(* CODESYS project partidas_v1_9_11.library
   DefaultNamespace: Teknike_Partidas
   DocFormat: reStructuredText
   Description: Bliblioteca com as partidas usadas pela Teknike
   Author: Tiago B. Cunico
   Title: Partidas
   Version: 1.9.11
   Company: Teknike
   Placeholder: Teknike_Partidas

Project tree, tasks and I/O mapping:
  libraries: OSCAT - AixOCAT, * (RWTH Aachen University - E.ON Energy Research Center); Tc2_MC2, * (Beckhoff Automation GmbH); Tc2_MC2_Drive, * (Beckhoff Automation GmbH); Tc2_ModbusRTU, * (Beckhoff Automation GmbH); Tc2_ModbusSrv, * (Beckhoff Automation GmbH); Tc2_Standard, * (Beckhoff Automation GmbH); Tc2_System, * (Beckhoff Automation GmbH); Tc2_Utilities, * (Beckhoff Automation GmbH); Tc3_Database, * (Beckhoff Automation GmbH); Tc3_Module, * (Beckhoff Automation GmbH); TcUnit, * (www.tcunit.org); Geral, * (Teknike)
  Legado/
    function block FB_ATV320CAN_V2_Legado [ST]: ACT_TrabalhaDados, ACT01_LeiturasCAN, ACT03_Cicla, ACT04_WriteCAN
    function block FB_Ethernet_ATV630_V2_Legado [ST]: ACT_00_LeituraETA_CIA402, ACT_01_LeituraVelocidadeAtual, ACT_03_EscritaVelocidade, ACT_04_Leitura_Last_error, ACT_05_LeituraETA_UINT, ACT_06_Leitura_Motor_Therm, ACT_07_Leitura_Motor_run_time, ACT_08_Leitura_Sto_Status, ACT_09_Leitura_APPS, ACT_HearthBeat
    function block FB_PartidaDireta_V2_Legado [ST]
    function block FB_PartidaDiretaReversao_V0_Legado [ST]
  POUs/
    Beckhoff/
      AX5000/
        Sts/
        function block FB_Comunicacao_AX5000 [ST]: ControlaACCDEC, LeParametros, Status
    Comunicação/
      CAN/
        Sts/
          data type ATV320_Can
          data type Config_CAN
          data type Config_CAN_Normal
          data type Config_CAN_Retentiva
          data type MaquinaCanOpen
        TeSys U/
          Sts/
            data type st_IosTeSysU_Can
            data type st_IosTeSysU_Can_IN
            data type st_IosTeSysU_Can_OUT
          function block FB_TeSysU_Can [ST]: AlertasEFalhas, IOs_vista
        function block FB_ComunicacaoCanOpen [ST]: AcaoMaquinaDeEstados, EscritaPDO, Escritas_SDO, Leituras_SDO, Status, TrocaEstadoMaquinaDeEstados
        function block SDO_READ [ST]
        function block SDO_WRITE [ST]
      Ethernet/
        data type ConfigComunicacaoEthernet
        function block ConversaoBilateralConfig [ST]
        function block FB_ComunicacaoEthernet [ST]: AcaoMaquinaDeEstados, Ciclo1s, Escrita, IHM, Leituras, Leituras_Escritas, MaquinaDeEstados, TrocaEstadoMaquinaDeEstados
        data type st_ReadWriteREG
      EthernetIP/
        Delta/
          Sts/
            data type st_LinkDeltaEIP
          function block FB_DeltaMS [ST]: ControleMarcha, ControleVelocidade, Emergencia, Others, Status
      ModbusRTU/
        STs/
          data type State_Modbus
          data type StateWord
        function block FB_ControleSoftRTU_LEGADO [ST]: Status
        function block FB_ModBusRTU_AC380 [ST]: Escrita, EspelhoEntradas, EspelhoSaidas, Estados, ExecutaEstados, Leitura, Leitura_Escrita, Status
        function block FB_ModBusRTU_ALTISTAR22 [ST]: Escrita, EspelhoEntradas, EspelhoSaidas, Estados, ExecutaEstados, Leitura, Leitura_Escrita, Status
        function block FB_ModBusRTU_ATV320 [ST]: Escrita, EspelhoEntradas, EspelhoSaidas, Estados, ExecutaEstados, Leitura, Leitura_Escrita, Status
    Partida/
      Sts/
        data type ST_ConfigInversor
        data type ST_ConfigMotorDB
        data type st_ConfigPartida
        data type st_EntradaPartida
        data type st_Erros
        data type st_KPIPartida
        data type st_LeiturasInversor
        data type st_LeiturasInversorIHM
        data type st_Partida
        data type st_SaidaPartida
      Test/
        function block FB_Partida_Teste [ST]: Bypasses, Emergencia, Falhas, Interlocks, ProxPartida, Reversao, Velocidade
      function block FB_Partida [ST]: AjustaEntradaST, AjustaSaida, AlarmesIHM, Contagem, ControleBloqueio, ControleDaPartida, ControleReset, ControleVelocidade, EmComissionamento, Falhas, FB_init, FirstScan, Horimetro, KPI, ProxMotor, SegurancaReversao, Status
    Siemens/
      Geral/
        data type bits
        data type Bits_8
        data type Duint
        data type Inversor_2Words_SinaSpeed
        data type InversorSinaSpeed
        data type sxRecvBuf
        data type sxSendBuf
        data type u16b
        data type Word_Bits
      SinaSpeed/
        data type EntradaSinaSpeed
        data type SaidaSinaSpeed
        function block Sina_SpeedV2 [ST]
        data type st_SinaSpeed
      function block Sina_posV2 [ST]
    global variables GVL_BlibliotecaPartidas
    program PRG_TEST [ST]: Teste, TesteAX5000, TesteCan, TesteCanTeSysU, TesteDelta, TestePartida, TestePartidaSimples, TesteProfinet
    program ValidaLicensa [ST]: Licensas
  Project Information/
    function F_GetCompany [ST]
    function F_GetTitle [ST]
    function F_GetVersion [ST]
  Version/
    global variables Global_Version
  VISUs/
*)

// POUs/Comunicação/CAN/Sts/ATV320_Can
TYPE ATV320_Can :
	STRUCT
		NodeState AT %I* : USINT;

		StatusWord		AT %I*	: UINT;
		ControlEffort	AT %I*	: INT;
		NM1				AT %I*	: UINT;
		NM2				AT %I*	: UINT;
		NM3				AT %I*	: UINT;
		NM4				AT %I*	: UINT;

		Controlword		AT %Q*	: UINT;
		TargetVelocity	AT %Q*	: INT;
		NC1				AT %Q*	: UINT;
		NC2				AT %Q*	: UINT;
		NC3				AT %Q*	: UINT;
		NC4				AT %Q*	: UINT;

	END_STRUCT
END_TYPE

// POUs/Comunicação/CAN/Sts/Config_CAN
TYPE Config_CAN :
	STRUCT
		Retentiva	: Config_CAN_Retentiva;
		Normal		: Config_CAN_Normal;
	END_STRUCT
END_TYPE

// POUs/Comunicação/CAN/Sts/Config_CAN_Normal
TYPE Config_CAN_Normal :
	STRUCT
		xLe				: BOOL;
		xEscreve_ITH	: BOOL;
		xEscreve_ACC	: BOOL;
		xEscreve_DEC	: BOOL;

		rITH_Lido	: REAL;
		rACC_Lido	: REAL;
		rDEC_Lido	: REAL;

	END_STRUCT
END_TYPE

// POUs/Comunicação/CAN/Sts/Config_CAN_Retentiva
TYPE Config_CAN_Retentiva :
STRUCT PERSISTENT RETAIN
	
	ACC_E 	: REAL;	//rampa de aceleração
	DEC_E 	: REAL;	//rampa de desaceleração
	
	NPR : REAL;
	NSP : REAL := 1800;
	NCR : REAL;
	ITH 	: REAL;	//corrente maxima 
	
	sAdressCAN		: STRING;	//Endereço CANOpen do Inversor em string
	wPortNrCAN		: WORD;		//numero da porta do inversor


END_STRUCT
END_TYPE

// POUs/Comunicação/CAN/Sts/MaquinaCanOpen
//{attribute 'qualified_only'}
{attribute 'strict'}
TYPE MaquinaCanOpen :
	(
		SwitchOnDisabled	:= 2,
		ReadyToSwitchOn		:= 3,
		SwitchedOn			:= 4,
		OperationEnabled	:= 5,
		QuickStopActive		:= 6,
		fault				:= 8
	);
END_TYPE

// POUs/Comunicação/CAN/TeSys U/Sts/st_IosTeSysU_Can
TYPE st_IosTeSysU_Can :
STRUCT
	en AT %I* : st_IosTeSysU_Can_IN;
	sa AT %Q* : st_IosTeSysU_Can_OUT;
	
	NodeState AT %I* : UsINT;
END_STRUCT
END_TYPE

// POUs/Comunicação/CAN/TeSys U/Sts/st_IosTeSysU_Can_IN
TYPE st_IosTeSysU_Can_IN :
STRUCT
	VarIn0 : WORD;//Control Register
	VarIn1 : WORD;//Control of communication module
	VarIn2 : WORD;//Output control
END_STRUCT
END_TYPE

// POUs/Comunicação/CAN/TeSys U/Sts/st_IosTeSysU_Can_OUT
TYPE st_IosTeSysU_Can_OUT :
STRUCT
	VarOut0 : WORD;//Status register
	VarOut1 : WORD;//I/O module status register
	VarOut2 : word;//Warning register
END_STRUCT
END_TYPE

// POUs/Comunicação/Ethernet/ConfigComunicacaoEthernet
TYPE ConfigComunicacaoEthernet :
	STRUCT
		rLSP				: REAL;	//velocidade minima
		rHSP				: REAL;	//velocidade maxima
		rTRF				: REAL;	//maxima velocidade
		rITH				: REAL;	//corrente maxima 
		rACC				: REAL;	//rampa de aceleração
		rDEC				: REAL;	//rampa de desaceleração
		xPHR				: BOOL;	//ordem das fases
		xEscreveParametros	: BOOL;
		xLerParametros		: BOOL;
		sIPAdress			: STRING(15); //Endereço Ethernet do Inversor
	END_STRUCT
END_TYPE

// POUs/Comunicação/Ethernet/st_ReadWriteREG
TYPE
	st_ReadWriteREG :
	STRUCT

		sIPAddr		: STRING;
		nQuantity	: WORD;
		nMBAddr		: WORD;
		cbLength	: UDINT;
		pDestAddr	: POINTER TO BYTE;
		xLe			: BOOL;
		xEscreve	: BOOL;
		nValue		: WORD;

		bBusy	: BOOL;
		bError	: BOOL;
		nErrID	: UDINT;
		cbRead	: UDINT;

	END_STRUCT
END_TYPE

// POUs/Comunicação/EthernetIP/Delta/Sts/st_LinkDeltaEIP
TYPE st_LinkDeltaEIP :
STRUCT
	state AT%I* : UINT;
	ErrorCode  AT%I* : UINT;
	iFrequenceCommand AT%I* : UINT;
	OutputFrequence AT%I* : UINT;
	OutputCurrent AT%I* : UINT;
	DCBusVoltage AT%I* : UINT;
	OutputVoltage AT%I* : UINT;
	Speed AT%I* : UINT;
	Counter AT%I* : UINT;
	IN_Value AT%I* : ARRAY[0..16] OF UINT;
	
	Control AT%Q* : UINT;
	oFrequenceCommand AT%Q* : UINT;
	Others AT%Q* : UINT;
	Out_Value AT%Q* : ARRAY[0..28] OF UINT;

END_STRUCT
END_TYPE

// POUs/Comunicação/ModbusRTU/STs/State_Modbus
{attribute 'qualified_only'}
{attribute 'strict'}
TYPE State_Modbus :
(
	Inicia			:= 0,
	Leitura			:= 1,
	Escrita			:= 2
);
END_TYPE

// POUs/Comunicação/ModbusRTU/STs/StateWord
{attribute 'qualified_only'}
{attribute 'strict'}
TYPE StateWord :
(
	LigacaoInibida		:= 0,
	NaoProntoParaLigar	:= 1,
	ProntoParaLigar		:= 2,
	OperacaoInibida		:= 3,
	ProntoParaOperar	:= 4,
	OperacaoAtiva		:= 5,
	SaidaAtivada		:= 6,
	AceleradorAtivos	:= 7,
	Operacao			:= 8,	
	Falha				:= 9,
	Off2				:= 10,
	Off3				:= 11					
);
END_TYPE

// POUs/Partida/Sts/ST_ConfigInversor
TYPE ST_ConfigInversor :
STRUCT RETAIN PERSISTENT
	ACC : REAL; // Rampa de aceleração
	xTemACC : BOOL; //Tem Rampa de aceleração
	DEC : REAL; // Rampa de desaceleração
	xTemDEC : BOOL; // Tem Rampa de desaceleração
	SuavidadeRampa : REAL; // se a rampa é mais de boa ou no tapao
	xTemSuavidadeRampa : BOOL; // Tem se a rampa é mais de boa ou no tapao
	ITH : REAL; // Corrente termica
	xTemITH : BOOL; //Tem Corrente termica
	HSP : REAL; // velocidade maxima
	xTemHSP : BOOL; //Tem velocidade maxima
	LSP : REAL; // velocidade minima
	xTemLSP : BOOL; //Tem velocidade minima
	BFR : REAL; // frequencia da rede
	xTemBFR : BOOL; //Tem frequencia da rede
	UNS : REAL; // tensao da rede
	xTemUNS : BOOL; //Tem tensao da rede
	NPR : REAL; // Potencia do motor
	xTemNPR : BOOL; //Tem Potencia do motor
	NCR : REAL; // Corrente do motor
	xTemNCR : BOOL; //Tem Corrente do motor
	NSP : REAL; // RPM do motor
	xTemNSP : BOOL; //Tem RPM do motor
	TFR : REAL; // Frequencia maxima do inversor
	xTemTFR : BOOL; //Tem Frequencia maxima do inversor
END_STRUCT
END_TYPE

// POUs/Partida/Sts/ST_ConfigMotorDB
TYPE ST_ConfigMotorDB :
STRUCT
	Motor: LINT;
	Tag: STRING(80);
	Funcao: STRING(80);
	InvIT1A: INT;
	IT1A: STRING(80);
	OPIT1: INT;
	InvIT1B: INT;
	IT1B: STRING(80);
	InvIT2A: INT;
	IT2A: STRING(80);
	OPIT2: INT;
	InvIT2B: INT;
	IT2B: STRING(80);
	InvIT3A: INT;
	IT3A: STRING(80);
	OPIT3: INT;
	InvIT3B: INT;
	IT3B: STRING(80);
	InvIT4A: INT;
	IT4A: STRING(80);
	OPIT4: INT;
	InvIT4B: INT;
	IT4B: STRING(80);
	Emerg1: STRING(80);
	Emerg2: STRING(80);
	Emerg3: STRING(80);
	Emerg4: STRING(80);
	Timestamp: DT;
END_STRUCT
END_TYPE

// POUs/Partida/Sts/st_ConfigPartida
TYPE st_ConfigPartida :
STRUCT RETAIN PERSISTENT
	
	inversor : ST_ConfigInversor;
	
	//Tempo para reversao sem tirar o comando de marcha
	xTemReversao			: BOOL;
	rTempoTrocaSentidoDeMarcha : REAL := 15;// esse tempo é pra evitar destruir a parte mecanica com a troca de sentido
	
	// Feedback da contatora
	rTempoFeedBackContator	: REAL := 1.5; (*Tempo entre acionar a Saída e receber o FeedBack da Contatora*)

	//Prox motor
	rTempoProxMotor			: REAL := 0.5;
	
	//Comissionamento
	xComissionado_Sentido : BOOL;
	xInverteSentido : BOOL; // bit pra inverrter o sentido do inversor

	//Conversao de velo em automatico
	xComissionado_Velo : BOOL;
	
	
	xVeloEmPorcentagem : BOOL; // usa o valor de 0-100% para controle da velo
	rVeloEmPorcentagem_VeloMax : REAL; // velo que representa 100%
	
	xVeloEmMetroPMin : BOOL; // usa a conversao para calcular a velocidade usada
	rVeloEmMetroPMin_Conversao : REAL; // valor em m/Min em 1000 RPM
	
	
	xComissionado_Corrente : BOOL;
	rCorrente_Comissionada : REAL;
	
	xTudoComissionado : BOOL;
	
	
	sNome_Funcao			:STRING;	// nome do motor e função para IHM
	rSetPoinAuto			:REAL;		// velocidadde que sera mandada para o bloco de comunicação
	rSetPoinAuto2			:REAL;		// velocidadde que sera mandada para o bloco de comunicação
	rSetPoinManu			:REAL;		// velocidadde que sera mandada para o bloco de comunicação
	xByPassContator			:BOOL;		//Sinal de by pass do contato da contatora
	xByPassDisjuntor		:BOOL;		//Sinal de by pass do contato do disjuntor

	xBypassRede				:BOOL;		// para caso tenha problema na rede ele poder operar sem ela
	
	xTemContatoInversorOK	:BOOL;		// esse cara é para o contado do inversor
	xBypassContatoInversorOK:BOOL;		// Bypass do xTemContatoInversorOK
		
	xBypassFreio 			: BOOL;		//bypass para o freio da partida
	xTemFreio 				: BOOL;		//variavel que diz que tem freio
	

	xTemSoft				: BOOL;		//Se tem soft			
	rTempoDeRampaSoft 		: REAL;		//Tempo pra rampa usando o contato de run dela pra finalizar a rampa
	xBypassContatoRunSoft 	: BOOL;		//bypass do contato de run dela
	xBypassContatoFalhaSoft : BOOL;		//bypass do contato de falha dela
	xBypassSoftEmFalhaCOM	: BOOL;		//Bypass da falha de comunicação
	
	xTemContatora			: BOOL;		// se tiver tru ele faz o esquema de ver se tem a contatora pra dar o erro se nao tiver feed back dela
	xTemDisjuntor			: BOOL;		// Pra caso nao tenha nao ficar dando erro
	
	
	xHabilitaHigienizacao	: BOOL; // Se tiver em true quando tiver xLigaHigienizacao ele vai ligar a esteira em rPorcentagemHigienizacao% da velo
	rPorcentagemHigienizacao: REAL;
	
	xTemLimiteReset 		: BOOL;//se a partida vai usar o limitador de reset
	iLimiteReset 			: INT;//Quantos reset pode dar antes de ter que dar o reset numero de reset
	iMinBloqueio			: ULINT;//por quantos minutos ele bloqueia antes de liberar sozinho o reset

	sIpInversor				: STRING;// Ip do inversor
	
END_STRUCT
END_TYPE

// POUs/Partida/Sts/st_EntradaPartida
TYPE
	st_EntradaPartida :
	STRUCT
		xEmergenciaOK		: BOOL;	(*Sinal de Emergência*)
		xContatorLigado		: BOOL;	(*Status da contatora ou do drive de que o motor partiu*)
		xDisjuntorOK		: BOOL;	(*Status do disjuntor motor*)
		xBloqueado			: BOOL;	//Sinal de Bloqueio
		iSenhaBloqueio		: INT;	//Senha de bloqueio
		iSenhaAtual			: INT;	// Senha que aparece no HMI
		xAutomaticoManual	: BOOL;	// se automatico = true se manual = false
		xLigaHigienizacao	: BOOL; // Quando acionado ele liga o motor em 10% da velo automatico
		xReversoAuto		: BOOL;	// habilita reverso em automatico
		xLigaAuto			: BOOL;	// liga inversor em automatico
		xUsaVeloAuto2		: BOOL; // Usa a segunda velo em automatico
		xReversoManu		: BOOL;	// liga inversor em manual
		xLigaManu			: BOOL;	// liga inversor em manual
		xLigaManu3S			: BOOL;	// Liga por 3 segundos em manual(Para comissionamento)
		xReset				: BOOL;	(*Sinal para resetar as falhas*)
		xResetRegistros		: BOOL;	(*Sinal apra resetar os contadores e registradores*)

		//Bloqueios
		xInterLock_1	: BOOL;		// sinal para bloquear a partida
		sInterLock_1	: STRING;	// porque o bloqueio 1
		xInterLock_2	: BOOL;		// sinal para bloquear a partida
		sInterLock_2	: STRING;	// porque o bloqueio 1
		xInterLock_3	: BOOL;		// sinal para bloquear a partida
		sInterLock_3	: STRING;	// porque o bloqueio 1
		xInterLock_4	: BOOL;		// sinal para bloquear a partida
		sInterLock_4	: STRING;	// porque o bloqueio 1

		//Inversor/comunicacao caso tenha
		xTemInversor			: BOOL;	// define se o bloco considera ou nao uma conexao
		xTemTeSysU				: BOOL; // Se tem TeSysU ele libera algumas informaçoes tipo a do inversor, mas nao libera tudo do inversor
		xInversorOnline			: BOOL;	// se etiver online
		xFalhaInversor			: BOOL;	// se o inversor tiver qualquer outra falha que nao seja perda de conexao
		xContatoInversorOK 		: BOOL; //Contato se o inversor esta OK
		xLocal					: BOOL; // caso o inversor esteja em modo local
		xResetBlocoComunicacao	: BOOL; //o reset do bloco vempor aqui, ai nao bate na contagem do reset
		xAlerta					: BOOL; //Status de alerta do inversor
		
		//horimetro
		stHoraAgora : TIMESTRUCT; // struct de hora para o horimetro

		i : INT; // index atual para a IHM

		xFazendoComissionamento : BOOL;

		xFreioOK : BOOL;
		
		xContatoFalhaSoft 	: BOOL;
		xContatoRodandoSoft : BOOL;
		xSoftEmFalhaCOM 	: BOOL;
		xSoftOnline 		: BOOL;
		
		iNumeroDeReset 		: INT;
		xResetaNumeroDeReset: BOOL;
		
		xECO : BOOL; //Entra no modo ECO - status igual a se estivesse com interlock
		
		xFaltaDeFaseOk : BOOL; // Se o falta de fase esta OK
		
		
	END_STRUCT
END_TYPE

// POUs/Partida/Sts/st_Erros
TYPE st_Erros :
STRUCT
	Mensagem 	: STRING;
	xErro		: BOOL;
	sTag		: STRING;
END_STRUCT
END_TYPE

// POUs/Partida/Sts/st_KPIPartida
TYPE st_KPIPartida :
	STRUCT
		
		stGraficoIHM : ARRAY[0..4] OF ST_Grafico;
		
		stGraficoOEE				: ARRAY[0..1] OF ST_Grafico;
		stGraficoDisponibilidade	: ARRAY[0..1] OF ST_Grafico;
		stGraficoPerformace			: ARRAY[0..1] OF ST_Grafico;
		stGraficoQualidade			: ARRAY[0..1] OF ST_Grafico;
	
		rPorcDesligado	: REAL;
		rPorcLigado		: REAL;
		rPorcInterlock	: REAL;
		rPorcFalha		: REAL;
		rPorcEmergencia	: REAL;

		tDesligado	: TIME;
		tLigado		: TIME;
		tInterlock	: TIME;
		tFalha		: TIME;
		tEmergencia	: TIME;
		
		iVezesDesligado 	: INT;
		iVezesLigado 		: INT;
		iVezesInterlock 	: INT;
		iVezesFalha 		: INT;
		iVezesEmergencia 	: INT;
		
		rDisponibilidade	: REAL;
		rPerformace			: REAL;
		rQualidade			: REAL := 100; // por padrao 100, mas se quiser forcar outro valor da
		rOEE				: REAL;
		
	END_STRUCT
END_TYPE

// POUs/Partida/Sts/st_LeiturasInversor
TYPE st_LeiturasInversor :
	STRUCT
		rVoltagemEntrada	: REAL;
		rTorque				: REAL;
		rTemperaturaInver	: REAL;
		rTemperaturaMotor	: REAL;
		rCorrente			: REAL;
		rVelocidadeRPM		: REAL;
		rVelocidadeHz		: REAL;
	END_STRUCT
END_TYPE

// POUs/Partida/Sts/st_LeiturasInversorIHM
TYPE st_LeiturasInversorIHM :
	STRUCT
		sVoltagemEntrada	: STRING;
		sTorque				: STRING;
		sTemperaturaInver	: STRING;
		sTemperaturaMotor	: STRING;
		sCorrente			: STRING;
		sVelocidadeRPM		: STRING;
		sVelocidadeHz		: STRING;
		sUltimoErro			: STRING;
		sStatusConexao		: STRING;
		
		xStatusEmergencias 	: ARRAY[1..4] OF BOOL;
		xStatusInterlocks 	: ARRAY[1..4,1..2] OF BOOL;	
	END_STRUCT
END_TYPE

// POUs/Partida/Sts/st_Partida
TYPE st_Partida :
	STRUCT
		En						: st_EntradaPartida;
		Sa						: st_SaidaPartida;
		LeiturasInversorIHM		: st_LeiturasInversorIHM;
		Config					: st_ConfigPartida;
		KPI						: ARRAY[0..23] OF st_KPIPartida;
		BancoDeDados			: ST_ConfigMotorDB;
		ErrosIHM				: ARRAY[0..20] OF st_Erros;
	END_STRUCT
END_TYPE

// POUs/Partida/Sts/st_SaidaPartida
TYPE st_SaidaPartida :
	STRUCT
		xLigado							: BOOL;	//sinal que o motor ta ligado, apesar de ele ter parado para fazer a reversao ou pelos interlocks
		xCmdFwd							: BOOL;	(*Liga Motor pra frente*)
		xCmdRev							: BOOL;	(*Liga Motor pra Tras*)
		xTrocandoSentido				: BOOL;	//quando ta trocando o sentido do motor ele deixa esse em true
		xParadoPorInterlock				: BOOL;	// se ele parar por algum interlock ele mostra aqui
		xTrocaReferenciaDeVelocidade	: BOOL;	// troca a referência de velocidade do inversor para local
		iVelocidade						: INT;	// velocidade para bloco de comunicação
		iStsMotor						: INT;	//olhas no action ststus para entender
		xResetParaInversor				: BOOL;	// sinal para o drive dar reset
		xFalha							: BOOL;	//Partida em falha
		xFalhaContatora 				: BOOL; //Sinal de falha da contatora para a IHM
		iDisjDesarm						: INT;	(*Contagem do numero de desarmes do disjuntor*)
		iPartidas						: INT;	(*Contagem do numero de partidas com sucesso do bloco*)
		iFalhaPartida					: INT;	(*Contagem do numero de falhas na partida do bloco*)

		// dados vindo do inversor, coloquei aqui para facilitar a visualização
		rVoltagemEntrada				: REAL;
		rTorque							: REAL;
		rTemperaturaInver				: REAL;
		rTemperaturaMotor				: REAL;
		rCorrente						: REAL;
		rVelocidadeRPM					: REAL;
		rVeloComissionada				: REAL;
		rVelocidadeHz					: REAL;
		sUltimoErro						: STRING;
		sAlerta							: STRING;
		sStatusConexao					: STRING;
		tHorimetro						: TIME;
		sHorimetro						: STRING;
		xNaoLigaProxMotor				: BOOL;
		
		sStatus 						: STRING;
	END_STRUCT
END_TYPE

// POUs/Siemens/Geral/bits
TYPE bits :
	STRUCT
		bBit0	: BIT;
		bBit1	: BIT;
		bBit2	: BIT;
		bBit3	: BIT;
		bBit4	: BIT;
		bBit5	: BIT;
		bBit6	: BIT;
		bBit7	: BIT;
		bBit8	: BIT;
		bBit9	: BIT;
		bBit10	: BIT;
		bBit11	: BIT;
		bBit12	: BIT;
		bBit13	: BIT;
		bBit14	: BIT;
		bBit15	: BIT;
	END_STRUCT
END_TYPE

// POUs/Siemens/Geral/Bits_8
TYPE Bits_8 :
	STRUCT
		bBit0	: BIT;
		bBit1	: BIT;
		bBit2	: BIT;
		bBit3	: BIT;
		bBit4	: BIT;
		bBit5	: BIT;
		bBit6	: BIT;
		bBit7	: BIT;
	END_STRUCT
END_TYPE

// POUs/Siemens/Geral/Duint
TYPE Duint :
	UNION
		Valor	: UDINT;
		uints	: ARRAY[0..1] OF UINT;
	END_UNION
END_TYPE

// POUs/Siemens/Geral/Inversor_2Words_SinaSpeed
TYPE Inversor_2Words_SinaSpeed :
	STRUCT
		StatusWord0	: u16b;
		StatusWord1	: u16b;
	END_STRUCT
END_TYPE

// POUs/Siemens/Geral/InversorSinaSpeed
TYPE InversorSinaSpeed :
	STRUCT
		StatusWord0		: u16b;
		StatusWord1		: u16b;
		StatusWord2		: u16b;
		StatusWord3		: u16b;
		StatusWord4		: u16b;
		StatusWord5		: u16b;
		StatusWord6		: u16b;
		StatusWord7		: u16b;
		StatusWord8		: u16b;
		StatusWord9		: u16b;
		StatusWord10	: u16b;
		StatusWord11	: u16b;
	END_STRUCT
END_TYPE

// POUs/Siemens/Geral/sxRecvBuf
TYPE sxRecvBuf :
	STRUCT
		ZSW1		: u16b;						//	Non-RETAIN	TRUE	TRUE	TRUE	FALSE	ZSW1sxZSW1         : STRUCT            NoFlwErr        : BOOL:=0;              // ZSW-Wort-1 Bit 08 --> 1 = Following error in tolerance            LbCr            : BOOL:=0;              // ZSW-Wort-1 Bit 09 --> 1 = Lifebit control request            TargPos         : BOOL:=0;              // ZSW-Wort-1 Bit 10 --> 1 = Target position reached            RefPSet         : BOOL:=0;              // ZSW-Wort-1 Bit 11 --> 1 = Reference point set            TrvTskAck       : BOOL:=0;              // ZSW-Wort-1 Bit 12 --> 1 = Traversing task acknowledge            StndStill       : BOOL:=0;              // ZSW-Wort-1 Bit 13 --> 1 = [n_ist] < Drehzahlsollwert 3            Accel           : BOOL:=0;              // ZSW-Wort-1 Bit 14 --> 1 = Axis accelerating            Decel           : BOOL:=0;              // ZSW-Wort-1 Bit 15 --> 1 = Axis decelerating            RTS             : BOOL:=0;              // ZSW-Wort-1 Bit 00 --> 1 = Ready to power up / to start            RDY             : BOOL:=0;              // ZSW-Wort-1 Bit 01 --> 1 = Ready to operate             IOp             : BOOL:=0;              // ZSW-Wort-1 Bit 02 --> 1 = In operation (operation enabled)            Fault           : BOOL:=0;              // ZSW-Wort-1 Bit 03 --> 1 = Fault present            NoOff2Act       : BOOL:=0;              // ZSW-Wort-1 Bit 04 --> 1 = OFF2 inactive            NoOff3Act       : BOOL:=0;              // ZSW-Wort-1 Bit 05 --> 1 = OFF3 inactive            PowInhbt        : BOOL:=0;              // ZSW-Wort-1 Bit 06 --> 1 = Power ON inhibit active             Alarm           : BOOL:=0;              // ZSW-Wort-1 Bit 07 --> 1 = Alarm / Warning present         END_STRUCT;
		EPosZSW1	: u16b;						//	Non-RETAIN	TRUE	TRUE	TRUE	FALSE	EPOSZSW1sxEPosZSW1     : STRUCT            StpCamMinAct    : BOOL:=0;              // EPOS-Wort-1 Bit 08 --> 1 = STOP cam minus active            StpCamPlsAct    : BOOL:=0;              // EPOS-Wort-1 Bit 09 --> 1 = STOP cam plus active            JogAct          : BOOL:=0;              // EPOS-Wort-1 Bit 10 --> 1 = Jogging active            RefAct          : BOOL:=0;              // EPOS-Wort-1 Bit 11 --> 1 = Reference point approach active            FlyRefAct       : BOOL:=0;              // EPOS-Wort-1 Bit 12 --> 1 = Flying referencing active            TrvBlAct        : BOOL:=0;              // EPOS-Wort-1 Bit 13 --> 1 = Traversing block active            MdiStupAct      : BOOL:=0;              // EPOS-Wort-1 Bit 14 --> 1 = MDI setup active            MdiPosAct       : BOOL:=0;              // EPOS-Wort-1 Bit 15 --> 1 = MDI positing active            ActTrvBit0      : BOOL:=0;              // EPOS-Wort-1 BIT 00 --> 1 = Active traversing block bit 0            ActTrvBit1      : BOOL:=0;              // EPOS-Wort-1 Bit 01 --> 1 = Active traversing block bit 1            ActTrvBit2      : BOOL:=0;              // EPOS-Wort-1 Bit 02 --> 1 = Active traversing block bit 2            ActTrvBit3      : BOOL:=0;              // EPOS-Wort-1 Bit 03 --> 1 = Active traversing block bit 3            ActTrvBit4      : BOOL:=0;              // EPOS-Wort-1 Bit 04 --> 1 = Active traversing block bit 4            ActTrvBit5      : BOOL:=0;              // EPOS-Wort-1 Bit 05 --> 1 = Active traversing block bit 5            Bit06           : BOOL:=0;              // EPOS-Wort-1 Bit 06 --> 1 = Reserve            Bit07           : BOOL:=0;              // EPOS-Wort-1 Bit 07 --> 1 = Reserve         END_STRUCT;
		EPosZSW2	: u16b;						//	Non-RETAIN	TRUE	TRUE	TRUE	FALSE	EPOSZSW2sxEPosZSW2      : STRUCT            PosSmCam1       : BOOL:=0;              // EPOS-Wort-2 Bit 08 --> 1 = Position actual value <= cam position 1            PosSmCam2       : BOOL:=0;              // EPOS-Wort-2 Bit 09 --> 1 = Position actual value <= cam position 2            TrvOut1         : BOOL:=0;              // EPOS-Wort-2 Bit 10 --> 1 = Direct output 1 via traversing block            TrvOut2         : BOOL:=0;              // EPOS-Wort-2 Bit 11 --> 1 = Direct output 2 via traversing block             FxStpRd         : BOOL:=0;              // EPOS-Wort-2 Bit 12 --> 1 = Fixed STOP reached            FxStpTrRd       : BOOL:=0;              // EPOS-Wort-2 Bit 13 --> 1 = Fixed STOP clamping torque reached            TrvFxStpAct     : BOOL:=0;              // EPOS-Wort-2 Bit 14 --> 1 = Traversing fixed STOP active            CmdAct          : BOOL:=0;              // EPOS-Wort-2 Bit 15 --> 1 = Traversing command active            TrkModeAct      : BOOL:=0;              // EPOS-Wort-2 Bit 00 --> 1 = Tracking mode active            VeloLimAct      : BOOL:=0;              // EPOS-Wort-2 Bit 01 --> 1 = Velocity limit active            SetPStat        : BOOL:=0;              // EPOS-Wort-2 Bit 02 --> 1 = Setpoint static            PrnMrkOut       : BOOL:=0;              // EPOS-Wort-2 Bit 03 --> 1 = Printmark outside outer window            FWD             : BOOL:=0;              // EPOS-Wort-2 Bit 04 --> 1 = Axis forwards            BWD             : BOOL:=0;              // EPOS-Wort-2 Bit 05 --> 1 = Axis backwards            SftSwMinAct     : BOOL:=0;              // EPOS-Wort-2 Bit 06 --> 1 = Software limit switch minus active            SftSwPlsAct     : BOOL:=0;              // EPOS-Wort-2 Bit 07 --> 1 = Software limit switch plus active         END_STRUCT;
		ZSW2		: u16b;						//	Non-RETAIN	TRUE	TRUE	TRUE	FALSE	ZSW2sxZSW2     : STRUCT            Bit08           : BOOL:=0;              // ZSW-Wort-2 Bit 08 --> Reserve            GlbTrgReq       : BOOL:=0;              // ZSW-Wort-2 Bit 09 --> Global trigger request            PulsEn          : BOOL:=0;              // ZSW-Wort-2 Bit 10 --> Pulses enabled            MotSwOverAct    : BOOL:=0;              // ZSW-Wort-2 Bit 11 --> Motor switch over activ            SlvZykBit0      : BOOL:=0;              // ZSW-Wort-2 Bit 12 --> Slave - life bit 0            SlvZykBit1      : BOOL:=0;              // ZSW-Wort-2 Bit 13 --> Slave - life bit 1            SlvZykBit2      : BOOL:=0;              // ZSW-Wort-2 Bit 14 --> Slave - life bit 2            SlvZykBit3      : BOOL:=0;              // ZSW-Wort-2 Bit 15 --> Slave - life bit 3            ActDDSBit0      : BOOL:=0;              // ZSW-Wort-2 Bit 00 --> Active drive data set bit 0            ActDDSBit1      : BOOL:=0;              // ZSW-Wort-2 Bit 01 --> Active drive data set bit 1            ActDDSBit2      : BOOL:=0;              // ZSW-Wort-2 Bit 02 --> Active drive data set bit 2            ActDDSBit3      : BOOL:=0;              // ZSW-Wort-2 Bit 03 --> Active drive data set bit 3            ActDDSBit4      : BOOL:=0;              // ZSW-Wort-2 Bit 04 --> Active drive data set bit 4            CmdActRelBrk    : BOOL:=0;              // ZSW-Wort-2 Bit 05 --> Command "release holding break" active            TrqContMode     : BOOL:=0;              // ZSW-Wort-2 Bit 06 --> Torque controlled mode            ParkAxisAct     : BOOL:=0;              // ZSW-Wort-2 Bit 07 --> Parking axis activated            END_STRUCT;
		NotUsed		: WORD := WORD#16#0000;		//	Non-RETAIN	TRUE	TRUE	TRUE	FALSE	Reserve
		Position	: duint;					//	Non-RETAIN	TRUE	TRUE	TRUE	FALSE	Feedback OF position
		Velocity	: duint;					//	Non-RETAIN	TRUE	TRUE	TRUE	FALSE	Feedback OF velocity
		ErrNr		: WORD	:= WORD#16#0000;	//	Non-RETAIN	TRUE	TRUE	TRUE	FALSE	Fault number
		WarnNr		: WORD	:= WORD#16#0000;	//	Non-RETAIN	TRUE	TRUE	TRUE	FALSE	Warning number
		Reserve		: WORD	:= WORD#16#0000;	//	Non-RETAIN	TRUE	TRUE	TRUE	FALSE	Reserve

	END_STRUCT
END_TYPE

// POUs/Siemens/Geral/sxSendBuf
TYPE sxSendBuf :
	STRUCT
		STW1		: u16b;						//Non-RETAIN	TRUE	TRUE	TRUE	FALSE	STW1sxSTW1     : STRUCT            Jog1            : BOOL:=0;              // ST-Wort-1 Bit 08 --> 1 = Jogging - signal source 1            Jog2            : BOOL:=0;              // ST-Wort-1 Bit 09 --> 1 = Jogging - signal source 2            LB              : BOOL:=1; // Allways   // ST-Wort-1 Bit 10 --> 1 = Life bit             RefStart        : BOOL:=0;              // ST-Wort-1 Bit 11 --> 1 = Referencing start / stop            Bit12           : BOOL:=0;              // ST-Wort-1 Bit 12 --> 1 = Reserve            Bit13           : BOOL:=0;              // ST-Wort-1 Bit 13 --> 1 = Externer Satzwechsel            Bit14           : BOOL:=0;              // ST-Wort-1 Bit 14 --> 1 = Reserve            Bit15           : BOOL:=0;              // ST-Wort-1 Bit 15 --> 1 = Reserve            Off1            : BOOL:=0;              // ST-Wort-1 Bit 00 --> 1 = OFF1/ON (flanks acceptance)            Off2            : BOOL:=1; // Allways   // ST-Wort-1 Bit 01 --> 1 = OFF2/ON (enable possible)            Off3            : BOOL:=1; // Allways   // ST-Wort-1 Bit 02 --> 1 = OFF3/ON (enable possible)            Enc             : BOOL:=1; // Allways   // ST-Wort-1 Bit 03 --> 1 = Enable controller            RejTrvTsk       : BOOL:=0;              // ST-Wort-1 Bit 04 --> 1 = Traversing block and MDI - reject task            IntMStop        : BOOL:=0;              // ST-Wort-1 Bit 05 --> 1 = Traversing block and MDI - intermediate - STOP            TrvStart        : BOOL:=0;              // ST-Wort-1 Bit 06 --> 1 = Traversing start - direct setpoint input / MDI - transfer edge            AckFault        : BOOL:=0;              // ST-Wort-1 Bit 07 --> 1 = Acknowledge fault         END_STRUCT;
		EPosSTW1	: u16b;						//Non-RETAIN	TRUE	TRUE	TRUE	FALSE	EPOSSTW1sxEPosSTW1   : STRUCT            MdiTyp          : BOOL:=0;              // EPOS-Wort-1 Bit 08 --> 1 = Direct setpoint input / MDI - positioning type            MdiPos          : BOOL:=0;              // EPOS-Wort-1 BIT 09 --> 1 = Direct setpoint input / MDI - positive direction            MdiNeg          : BOOL:=0;              // EPOS-Wort-1 BIT 10 --> 1 = Direct setpoint input / MDI - negative direction            Bit11           : BOOL:=0;              // EPOS-Wort-1 BIT 11 --> 1 = Reserve            MdiTrTyp        : BOOL:=0;              // EPOS-Wort-1 BIT 12 --> 1 = Direct setpoint input / MDI - transfer type            Bit13           : BOOL:=0;              // EPOS-Wort-1 BIT 13 --> 1 = Reserve            MdiSetup        : BOOL:=0;              // EPOS-Wort-1 BIT 14 --> 1 = Direct setpoint input / MDI - setup selection            MdiStart        : BOOL:=0;              // EPOS-Wort-1 BIT 15 --> 1 = Direct setpoint input / MDI - start              TrvBit0         : BOOL:=0;              // EPOS-Wort-1 BIT 00 --> 1 = Traversing block - block selection bit 0            TrvBit1         : BOOL:=0;              // EPOS-Wort-1 BIT 01 --> 1 = Traversing block - block selection bit 1            TrvBit2         : BOOL:=0;              // EPOS-Wort-1 BIT 02 --> 1 = Traversing block - block selection bit 2            TrvBit3         : BOOL:=0;              // EPOS-Wort-1 BIT 03 --> 1 = Traversing block - block selection bit 3            TrvBit4         : BOOL:=0;              // EPOS-Wort-1 BIT 04 --> 1 = Traversing block - block selection bit 4            TrvBit5         : BOOL:=0;              // EPOS-Wort-1 Bit 05 --> 1 = Traversing block - block selection bit 5            Bit06           : BOOL:=0;              // EPOS-Wort-1 Bit 06 --> 1 = Reserve            Bit07           : BOOL:=0;              // EPOS-Wort-1 Bit 07 --> 1 = Reserve          END_STRUCT;
		EPosSTW2	: u16b;						//Non-RETAIN	TRUE	TRUE	TRUE	FALSE	EPOSSTW2sxEPosSTW2   : STRUCT            RefTyp          : BOOL:=0;              // EPOS-Wort-2 Bit 08 --> 1 = Referencing type             RefStDi         : BOOL:=0;              // EPOS-Wort-2 Bit 09 --> 1 = Homing start direction            RefInpS         : BOOL:=0;              // EPOS-Wort-2 Bit 10 --> 1 = Referencing passive - input selection            RefEdge         : BOOL:=0;              // EPOS-Wort-2 Bit 11 --> 1 = Referencing passive - edge evaluation            Bit12           : BOOL:=0;              // EPOS-Wort-2 Bit 12 --> 1 = Reserve            Bit13           : BOOL:=0;              // EPOS-Wort-2 Bit 13 --> 1 = Reserve            SftLimAct       : BOOL:=0;              // EPOS-Wort-2 Bit 14 --> 1 = Software limit switch activation            StpCamAct       : BOOL:=0;              // EPOS-Wort-2 Bit 15 --> 1 = Stop output cam activation            TrkMode         : BOOL:=0;              // EPOS-Wort-2 Bit 00 --> 1 = Tracking mode active            SetRefPt        : BOOL:=0;              // EPOS-Wort-2 Bit 01 --> 1 = Set reference point            ActRefCam       : BOOL:=0;              // EPOS-Wort-2 Bit 02 --> 1 = Reference cam active            Bit03           : BOOL:=0;              // EPOS-Wort-2 Bit 03 --> 1 = Reserve            Bit04           : BOOL:=0;              // EPOS-Wort-2 Bit 04 --> 1 = Reserve            JogInc          : BOOL:=0;              // EPOS-Wort-2 Bit 05 --> 1 = Jogging - jogging incremental            Bit06           : BOOL:=0;              // EPOS-Wort-2 Bit 06 --> 1 = Reserve            Bit07           : BOOL:=0;              // EPOS-Wort-2 Bit 07 --> 1 = Reserve         END_STRUCT;
		STW2		: u16b;						//Non-RETAIN	TRUE	TRUE	TRUE	FALSE	STW2sxSTW2         : STRUCT            TrvFixStp       : BOOL:=0;              // ST-Wort-2 Bit 08 --> 1 = Travel fixed STOP            GlbTrgCom       : BOOL:=0;              // ST-Wort-2 Bit 09 --> 1 = Global trigger command            Bit10           : BOOL:=0;              // ST-Wort-2 Bit 10 --> 1 = Reserve            MotSwOver       : BOOL:=0;              // ST-Wort-2 Bit 11 --> 1 = Motor switch over finished            MsZykBit0       : BOOL:=0;              // ST-Wort-2 Bit 12 --> 1 = Master life bit 0            MsZykBit1       : BOOL:=0;              // ST-Wort-2 Bit 13 --> 1 = Master life bit 1            MsZykBit2       : BOOL:=0;              // ST-Wort-2 Bit 14 --> 1 = Master life bit 2            MsZykBit3       : BOOL:=0;              // ST-Wort-2 Bit 15 --> 1 = Master life bit 3            DDSBit0         : BOOL:=0;              // ST-Wort-2 Bit 00 --> 1 = Drive data set bit 0            DDSBit1         : BOOL:=0;              // ST-Wort-2 Bit 01 --> 1 = Drive data set bit 1            DDSBit2         : BOOL:=0;              // ST-Wort-2 Bit 02 --> 1 = Drive data set bit 2            DDSBit3         : BOOL:=0;              // ST-Wort-2 Bit 03 --> 1 = Drive data set bit 3            DDSBit4         : BOOL:=0;              // ST-Wort-2 Bit 04 --> 1 = Drive data set bit 4            GlbStart        : BOOL:=0;              // ST-Wort-2 Bit 05 --> 1 = Global start            ResIComp        : BOOL:=0;              // ST-Wort-2 Bit 06 --> 1 = Reset I-component of speed controller            ActPrkAxis      : BOOL:=0;              // ST-Wort-2 Bit 07 --> 1 = Activate parking axis            END_STRUCT;
		OverrideV	: WORD := WORD#16#0000;		//Non-RETAIN	TRUE	TRUE	TRUE	FALSE	Velocity override
		Position	: Duint;					//	Non-RETAIN	TRUE	TRUE	TRUE	FALSE	Setpoint OF position
		Velocity	: Duint;					//	Non-RETAIN	TRUE	TRUE	TRUE	FALSE	Setpoint OF velocity
		OverrideA	: WORD	:= WORD#16#0000;	//Non-RETAIN	TRUE	TRUE	TRUE	FALSE	Accelerating override
		OverrideD	: WORD	:= WORD#16#0000;	//Non-RETAIN	TRUE	TRUE	TRUE	FALSE	Decelerating override
		Reserve		: WORD	:= WORD#16#0000;	//Non-RETAIN	TRUE	TRUE	TRUE	FALSE	Reserve

	END_STRUCT
END_TYPE

// POUs/Siemens/Geral/u16b
TYPE u16b :
	UNION
		ui16b	: UINT;
		x16b	: bits;
	END_UNION
END_TYPE

// POUs/Siemens/Geral/Word_Bits
TYPE Word_Bits :
	UNION
		wor		: WORD;
		bits	: Bits_8;
	END_UNION
END_TYPE

// POUs/Siemens/SinaSpeed/EntradaSinaSpeed
TYPE EntradaSinaSpeed :
	STRUCT
		EnableAxis	: BOOL; //	0	Non-RETAIN	TRUE	TRUE	TRUE	FALSE	0-->1; 1 = Enable the drive (OFF2 / OFF 3 are 1 in default status) (OFF1 = 0-->1)
		AckError	:
			BOOL;						//	0	Non-RETAIN	TRUE	TRUE	TRUE	FALSE	1 = Acknowledge drive error
		SpeedSp			: REAL;			//	0.0	Non-retain	True	True	True	False	Speed standardises with the standardisation factor
		RefSpeed		: REAL;			//	0.0	Non-retain	True	True	True	False	Standardisation factor of speed
		ConfigAxis		: Word_Bits;	//	Non-RETAIN	TRUE	TRUE	TRUE	FALSE	binary programmed input TO control all functions in the telegram without its own FUNCTION block input
		HWIDZSW AT %I*	:
			InversorSinaSpeed; //	Non-retain	True	True	True	False	Hardware Identifer set point slot
	END_STRUCT
END_TYPE

// POUs/Siemens/SinaSpeed/SaidaSinaSpeed
TYPE SaidaSinaSpeed :
	STRUCT
		AxisEnabled	: BOOL;	//	0	Non-RETAIN	TRUE	TRUE	TRUE	FALSE	1 = Drive is enabled
		Lockout		: BOOL;	//	0	Non-RETAIN	TRUE	TRUE	TRUE	FALSE	1 = Drive lockout active
		ActVelocity	: REAL;	//	0.0	Non-RETAIN	TRUE	TRUE	TRUE	FALSE	Actual in [U/MIN]
		Error		: BOOL;	//	0	Non-RETAIN	TRUE	TRUE	TRUE	FALSE	1 = Error  (FB AND Infeed)
		Status		:
			WORD; //	0	Non-RETAIN	TRUE	TRUE	TRUE	FALSE	Status output (7002 = FB in operation; 8xxx = error description  - read the manual)
		DiagId :
			WORD; //	16#0000	Non-RETAIN	TRUE	TRUE	TRUE	FALSE	Error codes OF the cyclic system funtion blocks DPWR / DPRD_DAT
		HWIDSTW AT %Q* :
			Inversor_2Words_SinaSpeed; //	Non-retain	True	True	True	False	Hardware Identifer actual value slot
		Corrente	: REAL;
		Potencia	: REAL;
		Torque		: REAL;
		ErroAtual	: UINT;
	END_STRUCT
END_TYPE

// POUs/Siemens/SinaSpeed/st_SinaSpeed
TYPE st_SinaSpeed :
	STRUCT
		Entrada	: EntradaSInaSpeed;
		saida	: SaidaSinaSpeed;
	END_STRUCT
END_TYPE

// POUs/GVL_BlibliotecaPartidas
//{attribute 'qualified_only'}
VAR_GLOBAL
    {attribute 'hide'} 
	{attribute 'tc_no_symbol'}
	xLicensaValida5154156 : BOOL;
	LicensaValida : BOOL;
	STCheckLicense : ST_CheckLicense;
END_VAR

// Version/Global_Version
{attribute 'TcGenerated'}
{attribute 'no-analysis'}
{attribute 'linkalways'}
// This function has been automatically generated from the project information.
VAR_GLOBAL CONSTANT
	{attribute 'const_non_replaced'}
	stLibVersion_Partidas : ST_LibVersion := (iMajor := 1, iMinor := 9, iBuild := 11, iRevision := 0, nFlags := 0, sVersion := '1.9.11');
END_VAR

// Legado/FB_ATV320CAN_V2_Legado
FUNCTION_BLOCK FB_ATV320CAN_V2_Legado
VAR_INPUT
	xEnable					: BOOL;		//Sinal para Habilitar o Bloco de Controle
	xTipodeParada			: BOOL;		//Entrada para indicar o tipo da parada (0-Parada por rampa) (1-Parada por inércia)
	xParadaRapida			: BOOL;		//Entrada para parada rápida, quando acionado, o inversor força a parada rápida
	xResetDrive				: BOOL;		//Sinal de Entrada para Reset do Drive
	sAdressCAN				: STRING;	//Endereço CANOpen do Inversor em string
	wPortNrCAN				: WORD;		//numero da porta do inversor
	uiStatusWord			: UINT;
	xEmergencia				: BOOL; (*Sinal de Emergência*)
	xLiberadoOperar			: BOOL;
	xContatoInversor		: BOOL;
	xBypassContatoInversor	: BOOL;
	xDisjuntorMOTOR			: BOOL;
	xBypassDisjuntorMOTOR	: BOOL;
	iSetPoinAuto			: INT;
	iSetPoinManu			: INT;
	xAutomaticoManual		: BOOL;
	xLigaAuto				: BOOL;
	xDesligaAuto			: BOOL;
	xLigaManu				: BOOL;
	xDesligaManu			: BOOL;
	xSentidoReverso			: BOOL;
	xResetRegistros			: BOOL;
	xComecaLer				: BOOL;
END_VAR
VAR_OUTPUT
	xEnabled		: BOOL;	//Sinal de Saída que informa que o bloco está Habilitado		
	uiControlWord	: UINT;	//Control Word para o Inversor ATV320
	iTargetVelocity	: INT;	//Referencia de Velocidade para o inversor
	xResetInversor	: BOOL;	//Saída digital para Reset do inversor em caso de falha na rede
	uiFBState		: UINT;	//Variável que informa o estado do Bloco (1-Bloco Habilitado) (2-Nó CAN OK) (3-Nó CAN em Falha) (4- Inversor em RDY) (5-Falha na Energização do Drive) (6-Inversor em COF) (999-Bloco Desabilitado)
	xMotorRUN		: BOOL;	//Motor Rodando
	iStsWordHexa	: INT;	//ultimos dois digitos da Status Word do Inversor em Hexa
	rVeloHZ			: REAL;
	rMotorTorque	: REAL;
	rMotorCorrente	: REAL;
	iVeloRPM		: INT;
	iMotorVoltagem	: INT;
	iMotorPotencia	: INT;
	iMotorTemp		: INT;

	rVoltagemEntrada	: REAL;
	iInversorTemp		: INT;

	wStateWord			: WORD;
	sStatus				: STRING;
	xErroInversor		: BOOL;
	xWarningInversor	: BOOL;
	xReferenciaECont	: BOOL; //0 = display    1 = fildbus
	xSTOPInversor		: BOOL;
	xSentidoMotor		: BOOL; // 0 = frente	1 = reverso
	xInversorOnline		: BOOL;
	xCMDFwds			: BOOL;
	xFinalizou			: BOOL;
	istsMotor			: INT;
	iDisjDesarm			: INT;
	iPartidas			: INT;
	iInversoremFalha	: INT;
	dwStateColor		: DWORD;
	xInversoremFalha	: BOOL;
	xTerminouLeituras	: BOOL;
END_VAR
VAR
	xCmdFwd	: BOOL;	//Sinal digital para ligar o motor avanço
	xCmdRwd	: BOOL;	//Sinal digital para çigar o motor reverso

	xRedeCAN_OK			: BOOL;		//Flag que informa se a rede está OK
	xInversorRDY		: BOOL;		//Inversor em RDY
	iMachineState		: UINT;		//Controle da Máquina de Estado
	rtRedeOK			: R_TRIG;	//Indica que a rede Subiu
	ftRedeOK			: F_TRIG;	//Indica que a rede Caiu
	byteStatusWord		: BYTE;
	strHexStatusWord	: STRING;
	iStatusWordHexa		: INT;
	wETA				: WORD;
	sStatusTraducao		: ARRAY[1..15] OF STRING;

	ReadStart	: BOOL;
	ReadError	: DWORD;
	ReadData	: ARRAY[0..255] OF BYTE;

	SDO_READ		: ARRAY[1..14] OF SDO_READ;
	SDO_WRITE		: ARRAY[1..2] OF SDO_WRITE;
	xTerminouLer	: ARRAY[1..14] OF BOOL;
	fbCiclaLer		: FB_Ciclica;
	uiVolEntrada	: UINT;
	MainVoltage		: REAL;
	AuxLeitura		: UINT;
	rtComacaLeitura	: R_TRIG;
	i				: INT;

	xAuxNotOnline		: BOOL;
	rtComecaEscrever	: R_TRIG;
	xEscreveCMD			: BOOL;
	xEscreveVel			: BOOL;
	WriteDataVEL		: ARRAY[0..255] OF BYTE;
	WriteDataCTRL		: ARRAY[0..255] OF BYTE;

	iVelocidade : INT; //Entrada da referência de Velocidade

	rtIniciaMaquinadeEstados	: R_TRIG;
	rtNotOnline					: R_TRIG;
	tonOnline					: TON;

	(*Vai ficar aqui até decidir o que fazer com eles*)
	wCMDWord	: WORD;
	wSAF1		: WORD;

	Contador1				: CTU;
	Contador2				: CTU;
	Contador3				: CTU;
	wcont1					: WORD;
	wcont2					: WORD;
	wcont3					: WORD;
	FB_AnimaMotor			: FB_AnimaMotor;
	rtFalhanaPartida		: R_TRIG;
	rtSucessonaPartida		: R_TRIG;
	rtDisjuntorDesarmado	: R_TRIG;
	xFinalizou1				: BOOL;
	xFinalizou2				: BOOL;

	rtTrocouManAuto	: R_TRIG;
	ftTrocouManAuto	: F_TRIG;

END_VAR

IF xEnable THEN
	xEnabled := TRUE;
	ACT01_LeiturasCAN();
	ACT03_Cicla();
	ACT_TrabalhaDados();
	//	ACT04_WriteCAN();

	(*		
	uiFBState:=1;

(*Se o Nó estiver ativo, e sem falhas, energiza a potência do Drive*)
rtIniciaMaquinadeEstados(CLK:=xInversorOnline,Q=> );
	
	IF rtIniciaMaquinadeEstados.Q THEN
		iMachineState:=0;
	END_IF

	
IF iStatusWordHexa=17 AND NOT iMachineState=4 THEN  //535
	uiControlWord:= 0;	
END_IF


(*
IF iStatusWordHexa=33 AND NOT iMachineState=2 THEN
	iMachineState:= 2;	
END_IF
*)
*)

	rtTrocouManAuto(CLK := xAutomaticoManual, Q =>);
	ftTrocouManAuto(CLK := xAutomaticoManual, Q =>);

	IF rtTrocouManAuto.Q OR ftTrocouManAuto.Q THEN
		xCmdFWD	:= FALSE;
		xCmdRwd	:= FALSE;
	END_IF

	IF xEmergencia THEN
		IF xLiberadoOperar THEN
			IF ((xContatoInversor OR xBypassContatoInversor) AND (xDisjuntorMOTOR OR xBypassDisjuntorMOTOR)) THEN
				IF xAutomaticoManual THEN
					IF xLigaAuto THEN
						IF xSentidoReverso THEN
							xCmdRwd := TRUE;
						ELSE
							xCmdFWD := TRUE;
						END_IF
					END_IF

					IF xDesligaAuto THEN
						xCmdFWD	:= FALSE;
						xCmdRwd	:= FALSE;
					END_IF

					iVelocidade := iSetPoinAuto;
				ELSE // manual
					IF xLigaManu THEN
						IF xSentidoReverso THEN
							xCmdRwd := TRUE;
						ELSE
							xCmdFWD := TRUE;
						END_IF
					END_IF

					IF xDesligaManu THEN
						xCmdFWD	:= FALSE;
						xCmdRwd	:= FALSE;
					END_IF

					iVelocidade := iSetPoinManu;
				END_IF
			ELSE
				xCmdFWD	:= FALSE;
				xCmdRwd	:= FALSE;
			END_IF
		ELSE
			xCmdFWD	:= FALSE;
			xCmdRwd	:= FALSE;
		END_IF
	ELSE
		xCmdFWD	:= FALSE;
		xCmdRwd	:= FALSE;
	END_IF

	iTargetVelocity := iVelocidade;

	(*
//(*//comentado pelo bloco zuado
CASE iMachineState OF 

0:
	IF iStatusWordHexa=50 OR iStatusWordHexa=40  THEN //592
		uiControlWord:= 6; //Com o inversor em NST, joga o inversor para 'RDY'
	END_IF
	
	IF iStatusWordHexa=31 OR iStatusWordHexa=21 THEN //561
		iMachineState:=1; //com o inveror em RDY joga para o passo de ativação do comando
	END_IF
	
	IF iStatusWordHexa=33 THEN //563 ou 591
		iMachineState:=2; //com o inveror em RDY e ativado joga para o passo de comando
	END_IF
	
	
1:
	uiControlWord:= 7; //Com o inversor em RDY, Ativa o Comando
	
	IF iStatusWordHexa=33 THEN //563 ou 591
		iMachineState:=2; //com o inveror em RDY e ativado joga para o passo de comando
	END_IF
	
	IF iStatusWordHexa=50 THEN
		iMachineState:=0;
	END_IF
2:	

	IF iStatusWordHexa=50 THEN
		iMachineState:=0;
	END_IF

	IF uiControlWord= 15 AND iStatusWordHexa=33 AND NOT xCmdFwd THEN
		iMachineState:=1;
	END_IF


	IF xCmdFwd THEN 
		uiControlWord:= 15; //Comando de marcha avanço
		IF iStatusWordHexa=37 THEN
			iMachineState:=3;
		END_IF	
	END_IF

	IF xCmdRwd THEN 
		uiControlWord:= 2063; //Comando de marcha reverso
		IF iStatusWordHexa=37 THEN
			iMachineState:=5;
		END_IF	
	END_IF	
	
3:
IF iStatusWordHexa=37 THEN //1591
		IF NOT xCmdFwd THEN
			IF xTipodeParada THEN
			uiControlWord:= 7; //Comando de parada por rampa
			ELSE
			uiControlWord:= 6; //Comando de parada por inércia
			END_IF
		END_IF
		IF xParadaRapida THEN
			iMachineState:=4;		
		END_IF
END_IF

	IF iStatusWordHexa=31 THEN //561
		iMachineState:=1; //com o inveror em RDY joga para o passo de ativação do comando
	END_IF
	
	IF iStatusWordHexa=33 THEN //563
		iMachineState:=2; //com o inveror em RDY joga para o passo de ativação do comando
	END_IF
	
	IF iStatusWordHexa=50 THEN //592
		iMachineState:=6;
	END_IF	
	

4:
	uiControlWord:= 2; //Comando de parada rápida	
	
	IF iStatusWordHexa=17 THEN //535
		iMachineState:=0;
	END_IF

5:
IF iStatusWordHexa=37 THEN //34359
		IF NOT xCmdRwd THEN
			IF xTipodeParada THEN
			uiControlWord:= 7; //Comando de parada por rampa
			ELSE
			uiControlWord:= 6; //Comando de parada por inércia
			END_IF
		END_IF
		IF xParadaRapida THEN
			iMachineState:=4;		
		END_IF
END_IF

	IF iStatusWordHexa=31 THEN //561
		iMachineState:=1; //com o inveror em RDY joga para o passo de ativação do comando
	END_IF
	
	IF iStatusWordHexa=33 THEN //563
		iMachineState:=2; //com o inveror em RDY joga para o passo de ativação do comando
	END_IF
	
	IF iStatusWordHexa=50 THEN //592
		iMachineState:=6;
	END_IF	
	
6:
	uiControlWord:=0;
	IF 	iStatusWordHexa= 50 THEN
		iMachineState:=0;
	END_IF

	
ELSE
	uiControlWord:= 0; //Comando de parada rápida	

END_CASE

//Indica Motor Rodando Via Rede
IF iStatusWordHexa=37 THEN //1591
	xMotorRUN:=TRUE;
	ELSE
	xMotorRUN:=FALSE;
END_IF

IF iStatusWordHexa=50 THEN
	xMotorRUN:=FALSE;	
	IF xResetDrive THEN
		uiControlWord:= 128; //Comando de reset via rede	
	END_IF
END_IF


	ELSE
	uiControlWord:= 0;	//Se a rede CAN cair, joga o motor para parada por inércia 'NST'	
	xEnabled:= FALSE;
	uiFBState:=999;
	iMachineState:=0;
END_IF
//*)
//Copia sinal de liga para a saída do bloco
*)
END_IF

IF xResetDrive THEN
	//uiControlWord:= 128; //Comando de reset via rede
	xResetInversor := TRUE;
ELSE
	xResetInversor := FALSE;
END_IF

IF xContatoInversor THEN
	xCMDFwds := xCmdFWD;
ELSE
	xCMDFwds := FALSE;
END_IF

xAuxNotOnline := FALSE;

FOR i := 1 TO 14 DO
	IF SDO_READ[i].Error <> 0 THEN
		xAuxNotOnline := TRUE;
	END_IF
END_FOR

rtNotOnline(CLK := xAuxNotOnline, Q =>);
tonOnline(IN := NOT xAuxNotOnline, PT := T#3S, Q =>, ET =>);

IF rtNotOnline.Q THEN
	xInversorOnline := FALSE;
ELSIF tonOnline.Q THEN
	xInversorOnline := TRUE;
END_IF

IF (NOT xCmdFwd) AND xEmergencia THEN
	iStsMotor := 1;
END_IF

IF (xCmdFwd) AND xEmergencia THEN
	iStsMotor := 2;
END_IF

rtSucessonaPartida(CLK := (iStsMotor = 2), Q =>);

Contador2
	(
		CU := rtSucessonaPartida.Q,
			RESET := xResetRegistros,
			PV :=,
			Q =>,
			CV => wcont2);

IF (NOT xDisjuntorMOTOR) AND (NOT xBypassDisjuntorMOTOR) THEN
	iStsMotor := 3;
END_IF

rtDisjuntorDesarmado(CLK := iStsMotor = 3, Q =>);

Contador1
	(
		CU := rtDisjuntorDesarmado.Q,
			RESET := xResetRegistros,
			PV :=,
			Q =>,
			CV => wcont1);

//IF iStsWordHexa=38 OR NOT xInversorOnline THEN tirei pra nao dar erro quando nao online
IF iStsWordHexa = 38 THEN
	iStsMotor := 5;
END_IF

rtFalhanaPartida(CLK := iStsMotor = 5, Q =>);

Contador3
	(
		CU := rtFalhanaPartida.Q,
			RESET := xResetRegistros,
			PV :=,
			Q =>,
			CV => wcont3);

IF NOT xLiberadoOperar THEN
	iStsMotor := 6;
END_IF

IF NOT xEmergencia THEN
	iStsMotor := 4;
END_IF

iDisjDesarm			:= WORD_TO_INT(wcont1);
iPartidas			:= WORD_TO_INT(wcont2);
iInversoremFalha	:= WORD_TO_INT(wcont3);

FB_AnimaMotor(iStsMotor := iStsMotor, dwStateColor => dwStateColor);

ACTION ACT_TrabalhaDados:

sStatusTraducao[1]	:= 'Ready to switch on';
sStatusTraducao[2]	:= 'Switched on';
sStatusTraducao[3]	:= 'Running';
sStatusTraducao[4]	:= 'Erro detectado';
sStatusTraducao[5]	:= 'Warning';
sStatusTraducao[6]	:= 'referencia display';
sStatusTraducao[7]	:= 'referencia fildbus';
sStatusTraducao[8]	:= 'Stop local';
sStatusTraducao[9]	:= 'forward';
sStatusTraducao[10]	:= 'reverse';

xErroInversor		:= BIT_OF_DWORD(wETA, 3);
xWarningInversor	:= BIT_OF_DWORD(wETA, 7);
xReferenciaECont	:= BIT_OF_DWORD(wETA, 9);
xSTOPInversor		:= BIT_OF_DWORD(wETA, 14);
xSentidoMotor		:= BIT_OF_DWORD(wETA, 15);

//uiStatusWord:= WORD_TO_UINT(wETA);

(*Converte valor da Status Word para Hexa*)
byteStatusWord		:= UINT_TO_BYTE(uiStatusWord);
strHexStatusWord	:= BYTE_TO_HEXSTR(in := byteStatusWord, iPrecision := 2, bLoCase := FALSE);
iStatusWordHexa		:= STRING_TO_INT(strHexStatusWord);
iStsWordHexa		:= iStatusWordHexa;
(*---FIM---*)

IF NOT xInversorOnline THEN
	sStatus := 'Offline';
ELSE
	CASE iStsWordHexa OF
		31:
			sStatus				:= 'NST';
			xInversoremFalha	:= TRUE;

		33:
			sStatus				:= 'RDY';
			xInversoremFalha	:= FALSE;

		37:
			sStatus				:= 'RUN';
			xInversoremFalha	:= FALSE;

		38:
			sStatus				:= 'Falha';
			xInversoremFalha	:= TRUE;

		50:
			sStatus				:= 'STO / Emergencia';
			xInversoremFalha	:= TRUE;
	END_CASE
END_IF
END_ACTION

ACTION ACT01_LeiturasCAN:

rtComacaLeitura(CLK := xComecaLer, Q =>);

IF rtComacaLeitura.Q THEN
	xTerminouLer[1]		:= TRUE;
	xTerminouLeituras	:= FALSE;
END_IF

////////////////// voltagem de entrada///////////////////////////

SDO_READ[1]
	(
		StartReading := xTerminouLer[1],
			CO_Index := 16#2002,
			CO_SubIndex := 16#8,
			DataLength := SIZEOF(UINT),
			PortNr := wPortNrCAN,
			ADSNetID := sAdressCAN);

IF SDO_READ[1].ReadDataAvailable AND xTerminouLer[1] THEN
	xComecaLer		:= FALSE;
	xTerminouLer[1]	:= FALSE;
	xTerminouLer[2]	:= TRUE;
	ReadError		:= SDO_READ[1].Error;
	ReadData		:= SDO_READ[1].ReadData;
	MEMCPY(destAddr := ADR(AuxLeitura), srcAddr := ADR(ReadData), n := SIZEOF(UINT));
	rVoltagemEntrada := UINT_TO_REAL(AuxLeitura) / 10;
END_IF

////////////////// Velo em Hz///////////////////////////
SDO_READ[2]
	(
		StartReading := xTerminouLer[2],
			CO_Index := 16#2002,
			CO_SubIndex := 16#3,
			DataLength := SIZEOF(UINT),
			PortNr := wPortNrCAN,
			ADSNetID := sAdressCAN);

IF SDO_READ[2].ReadDataAvailable AND xTerminouLer[2] THEN
	xTerminouLer[2]	:= FALSE;
	xTerminouLer[3]	:= TRUE;

	ReadError	:= SDO_READ[2].Error;
	ReadData	:= SDO_READ[2].ReadData;
	MEMCPY(destAddr := ADR(AuxLeitura), srcAddr := ADR(ReadData), n := SIZEOF(UINT));
	rVeloHZ := UINT_TO_REAL(AuxLeitura) / 10;
END_IF

////////////////// Velo em RPM///////////////////////////
SDO_READ[3]
	(
		StartReading := xTerminouLer[3],
			CO_Index := 16#2038,
			CO_SubIndex := 16#5,
			DataLength := SIZEOF(UINT),
			PortNr := wPortNrCAN,
			ADSNetID := sAdressCAN);

IF SDO_READ[3].ReadDataAvailable AND xTerminouLer[3] THEN
	xTerminouLer[3]	:= FALSE;
	xTerminouLer[4]	:= TRUE;
	ReadError		:= SDO_READ[3].Error;
	ReadData		:= SDO_READ[3].ReadData;
	MEMCPY(destAddr := ADR(AuxLeitura), srcAddr := ADR(ReadData), n := SIZEOF(UINT));
	iVeloRPM := UINT_TO_INT(AuxLeitura);

END_IF

////////////////// Corrente Motor///////////////////////////
SDO_READ[4]
	(
		StartReading := xTerminouLer[4],
			CO_Index := 16#2002,
			CO_SubIndex := 16#5,
			DataLength := SIZEOF(UINT),
			PortNr := wPortNrCAN,
			ADSNetID := sAdressCAN);

IF SDO_READ[4].ReadDataAvailable AND xTerminouLer[4] THEN
	xTerminouLer[4]	:= FALSE;
	xTerminouLer[5]	:= TRUE;
	ReadError		:= SDO_READ[4].Error;
	ReadData		:= SDO_READ[4].ReadData;
	MEMCPY(destAddr := ADR(AuxLeitura), srcAddr := ADR(ReadData), n := SIZEOF(UINT));
	rMotorCorrente := UINT_TO_REAL(AuxLeitura) / 10;
END_IF

////////////////// Potencia do motor ///////////////////////////
SDO_READ[5]
	(
		StartReading := xTerminouLer[5],
			CO_Index := 16#2002,
			CO_SubIndex := 16#C,
			DataLength := SIZEOF(UINT),
			PortNr := wPortNrCAN,
			ADSNetID := sAdressCAN);

IF SDO_READ[5].ReadDataAvailable AND xTerminouLer[5] THEN
	xTerminouLer[5]	:= FALSE;
	xTerminouLer[6]	:= TRUE;
	ReadError		:= SDO_READ[5].Error;
	ReadData		:= SDO_READ[5].ReadData;
	MEMCPY(destAddr := ADR(AuxLeitura), srcAddr := ADR(ReadData), n := SIZEOF(UINT));
	iMotorPotencia := UINT_TO_INT(AuxLeitura);
END_IF

//////////////////Temperatura do inversor///////////////////////////
SDO_READ[6]
	(
		StartReading := xTerminouLer[4],
			CO_Index := 16#2002,
			CO_SubIndex := 16#A,
			DataLength := SIZEOF(UINT),
			PortNr := wPortNrCAN,
			ADSNetID := sAdressCAN);

IF SDO_READ[6].ReadDataAvailable AND xTerminouLer[6] THEN
	xTerminouLer[6]	:= FALSE;
	xTerminouLer[7]	:= TRUE;
	ReadError		:= SDO_READ[6].Error;
	ReadData		:= SDO_READ[6].ReadData;
	MEMCPY(destAddr := ADR(AuxLeitura), srcAddr := ADR(ReadData), n := SIZEOF(UINT));
	iInversorTemp := UINT_TO_INT(AuxLeitura);
END_IF

////////////////// Temperatura do motor///////////////////////////
SDO_READ[7]
	(
		StartReading := xTerminouLer[7],
			CO_Index := 16#2042,
			CO_SubIndex := 16#1F,
			DataLength := SIZEOF(UINT),
			PortNr := wPortNrCAN,
			ADSNetID := sAdressCAN);

IF SDO_READ[7].ReadDataAvailable AND xTerminouLer[7] THEN
	xTerminouLer[7]	:= FALSE;
	xTerminouLer[8]	:= TRUE;
	ReadError		:= SDO_READ[7].Error;
	ReadData		:= SDO_READ[7].ReadData;
	MEMCPY(destAddr := ADR(AuxLeitura), srcAddr := ADR(ReadData), n := SIZEOF(UINT));
	iMotorTemp := UINT_TO_INT(AuxLeitura);
END_IF

////////////////// State Word///////////////////////////
SDO_READ[8]
	(
		StartReading := xTerminouLer[8],
			CO_Index := 16#202A,
			CO_SubIndex := 16#B,
			DataLength := SIZEOF(WORD),
			PortNr := wPortNrCAN,
			ADSNetID := sAdressCAN);

IF SDO_READ[8].ReadDataAvailable AND xTerminouLer[8] THEN
	xTerminouLer[8]	:= FALSE;
	xTerminouLer[9]	:= TRUE;
	ReadError		:= SDO_READ[8].Error;
	ReadData		:= SDO_READ[8].ReadData;
	MEMCPY(destAddr := ADR(AuxLeitura), srcAddr := ADR(ReadData), n := SIZEOF(WORD));
	wStateWord := AuxLeitura;
END_IF

////////////////// Comand Word///////////////////////////
SDO_READ[9]
	(
		StartReading := xTerminouLer[9],
			CO_Index := 16#202A,
			CO_SubIndex := 16#1F,
			DataLength := SIZEOF(WORD),
			PortNr := wPortNrCAN,
			ADSNetID := sAdressCAN);

IF SDO_READ[9].ReadDataAvailable AND xTerminouLer[9] THEN
	xTerminouLer[9]		:= FALSE;
	xTerminouLer[10]	:= TRUE;
	ReadError			:= SDO_READ[9].Error;
	ReadData			:= SDO_READ[9].ReadData;
	MEMCPY(destAddr := ADR(AuxLeitura), srcAddr := ADR(ReadData), n := SIZEOF(WORD));
	wCMDWord := AuxLeitura;
END_IF

////////////////// Saf1 app Safety///////////////////////////
SDO_READ[10]
	(
		StartReading := xTerminouLer[10],
			CO_Index := 16#207B,
			CO_SubIndex := 16#33,
			DataLength := SIZEOF(WORD),
			PortNr := wPortNrCAN,
			ADSNetID := sAdressCAN);

IF SDO_READ[10].ReadDataAvailable AND xTerminouLer[10] THEN
	xTerminouLer[10]	:= FALSE;
	xTerminouLer[11]	:= TRUE;
	ReadError			:= SDO_READ[10].Error;
	ReadData			:= SDO_READ[10].ReadData;
	MEMCPY(destAddr := ADR(AuxLeitura), srcAddr := ADR(ReadData), n := SIZEOF(WORD));
	wSAF1 := AuxLeitura;
END_IF

////////////////// Drivecom state register ETA///////////////////////////
SDO_READ[11]
	(
		StartReading := xTerminouLer[11],
			CO_Index := 16#2002,
			CO_SubIndex := 16#2,
			DataLength := SIZEOF(WORD),
			PortNr := wPortNrCAN,
			ADSNetID := sAdressCAN);

IF SDO_READ[11].ReadDataAvailable AND xTerminouLer[11] THEN
	xTerminouLer[11]	:= FALSE;
	xComecaLer			:= FALSE;
	//		xTerminouLer[12] := TRUE;
	xTerminouLeituras	:= TRUE;
	ReadError			:= SDO_READ[11].Error;
	ReadData			:= SDO_READ[11].ReadData;
	MEMCPY(destAddr := ADR(AuxLeitura), srcAddr := ADR(ReadData), n := SIZEOF(WORD));
	wETA := AuxLeitura;
END_IF
END_ACTION

ACTION ACT03_Cicla:
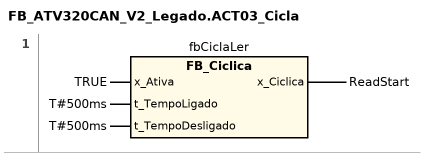
// NETWORK 1
fbCiclaLer(x_Ativa := TRUE, t_TempoLigado := T#500ms, t_TempoDesligado := T#500ms); // FB_Ciclica
ReadStart := fbCiclaLer.x_Ciclica;
END_ACTION

ACTION ACT04_WriteCAN:
//rtComecaEscrever(CLK:= ReadStart, Q=> );

//IF rtComecaEscrever.Q THEN	
//	xEscreveCMD := TRUE;
//	xEscreveVel := TRUE;
//	xFinalizou1 := FALSE;
//	xFinalizou2 := FALSE;
//END_IF

// converte Control Word de UINT para byte array
MEMCPY(destAddr := ADR(WriteDataCTRL), srcAddr := ADR(uiControlWord), n := SIZEOF(WriteDataCTRL));

//Escreve a Control Word no Inversor
SDO_WRITE[1]
	(
		ADSNetID := sAdressCAN,
			PortNr := wPortNrCAN,
			CO_Index := 16#2037,
			CO_SubIndex := 16#2,
			DataLength := SIZEOF(WORD),
			StartWriting := xTerminouLer[12],
			WriteData := WriteDataCTRL,
			WriteDataFinished =>,
			Error =>);

IF SDO_WRITE[1].WriteDataFinished AND xTerminouLer[12] THEN
	xTerminouLer[12]	:= FALSE;
	xTerminouLer[13]	:= TRUE;
END_IF

// converte velocidade de int para byte array
MEMCPY(destAddr := ADR(WriteDataVEL), srcAddr := ADR(iTargetVelocity), n := SIZEOF(WriteDataVEL));

//Escreve a Velocidade no Inversor	
SDO_WRITE[2]
	(
		ADSNetID := sAdressCAN,
			PortNr := wPortNrCAN,
			CO_Index := 16#2038,
			CO_SubIndex := 16#3,
			DataLength := SIZEOF(WORD),
			StartWriting := xTerminouLer[13],
			WriteData := WriteDataVEL,
			WriteDataFinished =>,
			Error =>);

IF SDO_WRITE[2].WriteDataFinished AND xTerminouLer[13] THEN
	xTerminouLer[13]	:= FALSE;
	xTerminouLeituras	:= TRUE;
END_IF

xFinalizou := xFinalizou1 AND xFinalizou2;
END_ACTION

END_FUNCTION_BLOCK

// POUs/Comunicação/CAN/SDO_READ
FUNCTION_BLOCK SDO_READ
VAR_INPUT
	ADSNetID : STRING(23); (* The AMSNetID addresses the EL6751. Can be empty if only one local single cha
nnel card is present*)
	PortNr			: WORD;		(* This Port No. addresses the CANopen Node (see System Manager) *)
	CO_Index		: DWORD;	(* This is the Index of the CANopen Object Dictionary Entry*)
	CO_SubIndex		: DWORD;	(* This is the Sub-Index of the CANopen Object Dictionary Entry*)
	DataLength		: DWORD;	(* This is the Length of the CANopen Object Dictionary Entry*)
	StartReading	: BOOL;		(* only reset to FALSE after ReadDataAvailable=TRUE*)
END_VAR
VAR_OUTPUT
	ReadData			: ARRAY[0..255] OF BYTE;
	ReadDataAvailable	: BOOL;
	Error				: DWORD;
END_VAR
VAR
	state	: BYTE := 0;
	ADSREAD	: ADSREAD;
END_VAR


IF xLicensaValida5154156 THEN
	
	
	CASE
		state OF
		0:
			IF StartReading THEN
				ReadDataAvailable	:= FALSE;
				Error				:= 0;
	
				ADSRead
					(
						NETID := ADSNetID,
							PORT := PortNr,
							IDXGRP := CO_Index,
							IDXOFFS := CO_SubIndex,
							LEN := DataLength,
							DESTADDR := ADR(ReadData),
							READ := TRUE,
							TMOUT := T#1S);
	
				IF ADSRead.err THEN
					state				:= 2;
					ReadDataAvailable	:= TRUE;
					Error				:= ADSRead.ErrId;
				ELSE
					state := 1;
				END_IF
			ELSE
				ADSRead
					(
						NETID := ADSNetID,
							PORT := PortNr,
							IDXGRP := CO_Index,
							IDXOFFS := CO_SubIndex,
							LEN := DataLength,
							DESTADDR := ADR(ReadData),
							READ := FALSE,
							TMOUT := T#1s);
			END_IF
	
		1:
			ADSRead(READ := FALSE);
	
			IF ADSRead.err THEN
				state				:= 2;
				ReadDataAvailable	:= TRUE;
				Error				:= ADSRead.ErrId;
			ELSE
				IF NOT ADSRead.busy THEN
					state				:= 2;
					ReadDataAvailable	:= TRUE;
				END_IF
			END_IF
	
		2:
			ADSRead(READ := FALSE);
			state := 0;
	END_CASE

ELSE
	ValidaLicensa();
END_IF

END_FUNCTION_BLOCK

// POUs/ValidaLicensa
PROGRAM ValidaLicensa
VAR
{attribute 'tc_no_symbol'}
Olhaliscensa : FB_CheckLicense;
{attribute 'tc_no_symbol'}
GUIDLicensa : GUID := STRING_TO_GUID('17F8A500-35EB-4504-A538-37BC9FA779F1');
END_VAR


Licensas();

STCheckLicense := Olhaliscensa.stCheckLicense;

xLicensaValida5154156 :=
 Olhaliscensa.stCheckLicense.eResult = 0 OR
 Olhaliscensa.stCheckLicense.eResult = 16#203 OR
 Olhaliscensa.stCheckLicense.eResult = 16#254 OR
 Olhaliscensa.stCheckLicense.eResult = 16#255;

 LicensaValida := xLicensaValida5154156;

ACTION Licensas:
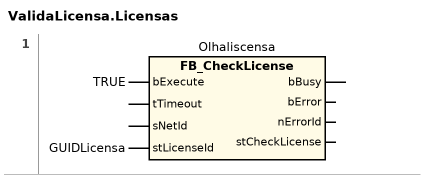
// NETWORK 1
Olhaliscensa(bExecute := TRUE, stLicenseId := GUIDLicensa); // FB_CheckLicense
END_ACTION

END_PROGRAM

// POUs/Comunicação/CAN/SDO_WRITE
FUNCTION_BLOCK SDO_WRITE
VAR_INPUT
	ADSNetID : STRING(23); (* The AMSNetID addresses the EL6751. Can be empty if only one local single c
hannel card is present*)
	PortNr			: WORD;						(* The Port No. addresses the CANopen Node (see System Manager) *)
	CO_Index		: DWORD;					(* This is the Index of the CANopen Object Dictionary Entry*)
	CO_SubIndex		: DWORD;					(*This is the Sub-Index of the CANopen Object Dictionary Entry*)
	DataLength		: DWORD;					(* This is the Length of the CANopen Object Dictionary Entry*)
	StartWriting	: BOOL;						(*only reset to FALSE after WriteDataFinished=TRUE*)
	WriteData		: ARRAY[0..255] OF BYTE;	(*This array contains the data to be written to the CANopen Object
Dictionary*)
END_VAR
VAR_OUTPUT
	WriteDataFinished	: BOOL;
	Error				: DWORD;
END_VAR
VAR
	state		: BYTE := 0;
	ADSWRITE	: ADSWRITE;
END_VAR

IF xLicensaValida5154156 THEN

	
	CASE
		state OF
		0:
			IF StartWriting THEN
				WriteDataFinished	:= FALSE;
				Error				:= 0;
	
				ADSWrite
					(
						NETID := ADSNetID,
							PORT := PortNr,
							IDXGRP := CO_Index,
							IDXOFFS := CO_SubIndex,
							LEN := DataLength,
							SRCADDR := ADR(WriteData),
							WRITE := TRUE,
							TMOUT := T#1s);
	
				IF ADSWrite.err THEN
					state				:= 2;
					WriteDataFinished	:= TRUE;
					Error				:= ADSWrite.ErrId;
				ELSE
					state := 1;
				END_IF
			ELSE
				ADSWrite
					(
						NETID := '',
							PORT := PortNr,
							IDXGRP := CO_Index,
							IDXOFFS := CO_SubIndex,
							LEN := DataLength,
							SRCADDR := ADR(WriteData),
							WRITE := FALSE,
							TMOUT := T#1s);
			END_IF
	
		1:
			ADSWrite(WRITE := FALSE);
	
			IF ADSWrite.err THEN
				state				:= 2;
				WriteDataFinished	:= TRUE;
				Error				:= ADSWrite.ErrId;
			ELSE
				IF NOT ADSWrite.busy THEN
					state				:= 2;
					WriteDataFinished	:= TRUE;
				END_IF
			END_IF
	
		2:
			ADSWrite(WRITE := FALSE);
			state := 0;
	END_CASE

ELSE
	ValidaLicensa();
END_IF

END_FUNCTION_BLOCK

// Legado/FB_Ethernet_ATV630_V2_Legado
FUNCTION_BLOCK FB_Ethernet_ATV630_V2_Legado
VAR_INPUT
	xEnable			: BOOL;			//Sinal para Habilitar o Bloco de Controle
	xTipodeParada	: BOOL;			//Entrada para indicar o tipo da parada (0-Parada por rampa) (1-Parada por inércia)
	xParadaRapida	: BOOL;			//Entrada para parada rápida, quando acionado, o inversor força a parada rápida
	xResetDrive		: BOOL;			//Sinal de Entrada para Reset do Drive
	sIPAdress		: STRING(15);	//Endereço Ethernet do Inversor
	// add 08/10/2020 por Tiago
	xDisjuntorMOTOR			: BOOL;	// SInal do Disjuntor MOTOR
	xBypassDisjuntorMOTOR	: BOOL;	//Bypass do sinal do Disjuntor MOTOR
	xContatoInversor		: BOOL;	//Sinal do contato do inversor
	xBypassContatoInversor	: BOOL;	//Bypass do sinal do contato do inversor
	xEmergencia				: BOOL;	(*Sinal de Emergência*)
	xLiberadoOperar			: BOOL;
	xLigaAuto				: BOOL;	// liga inversor em automatico
	xDesligaAuto			: BOOL;	// Desliga inversor em automatico
	xLigaManu				: BOOL;	// liga inversor em manual
	xDesligaManu			: BOOL;	// Desliga inversor em manual
	xAutomaticoManual		: BOOL;	// se automatico = true se manual = false
	iSetPoinManu			: INT;	// set point do manual
	iSetPoinAuto			: INT;	// set point do auto
	xSentidoReverso			: BOOL;
	xResetRegistros			: BOOL;

END_VAR
VAR_OUTPUT
	xEnabled				: BOOL;		//Sinal de Saída que informa que o bloco está Habilitado		
	uiControlWord			: UINT;		//Control Word para o Inversor ATV320
	iTargetVelocity			: INT;		//Referencia de Velocidade para o inversor
	xResetInversor			: BOOL;		//Saída digital para Reset do inversor em caso de falha na rede
	uiFBState				: UINT;		//Variável que informa o estado do Bloco (1-Bloco Habilitado) (2-Nó CAN OK) (3-Nó CAN em Falha) (4- Inversor em RDY) (5-Falha na Energização do Drive) (6-Inversor em COF) (999-Bloco Desabilitado)
	xMotorRUN				: BOOL;		//Motor Rodando
	iStsWordHexa			: INT;		//ultimos dois digitos da Status Word do Inversor em Hexa
	iVelocidadeAtual		: INT;		//Retorno da velocidade real do inversor
	rCorrenteAtual			: REAL;		//Corrente Atual no Motor
	rVelocidadeAtualHZ		: REAL;		//Velocidade Atual no motor em HZ
	iMotorTorqueAtual		: INT;		//Torque atual do motor
	iMotorVoltagemAtual		: INT;		//Voltagem atual do motor
	rVoltagemEntrada		: REAL;		//Voltagem atual na entrada
	rTemperaturaInversor	: REAL;		//Temperatura atual no inversor em %
	iLastError				: INT;		//Codigo do ultimo erro
	iTemperaturaMotorAtual	: INT;		//Temperatura do motor atual em %
	iTempoMotorLigadoSempre	: UINT;		// tempo em segundos que o motor esteve ligado desde sempre, nao reinicia apos desligar
	xStatusEmergencia		: BOOL;		// status do sto
	sStatusInversor			: STRING;	// status do inversor
	tTempoLigadoAgora		: TIME;		// tempo que o inversor esta ligado desde a ultima parada
	// add 08/10/2020 por Tiago
	xInversorOnline		: BOOL;		// se inversor online
	xCMDFwds			: BOOL;		// sinal para controle do inversor sem ethernet
	sWordTraduzida		: STRING;	// string da word de status traduzida
	istsMotor			: INT;
	iDisjDesarm			: INT;
	iPartidas			: INT;
	iInversoremFalha	: INT;
	dwStateColor		: DWORD;
	xInversoremFalha	: BOOL;
END_VAR
VAR
	//xRedeCAN_OK		: BOOL;		//Flag que informa se a rede está OK
	xInversorRDY		: BOOL;		//Inversor em RDY
	iMachineState		: INT;		//Controle da Máquina de Estado
	rtWriteCtrlWord		: R_TRIG;	//necessidade de escrever a Ctrl Word
	rtWriteSpeed		: R_TRIG;	//Necessidade de escrever a velocidade
	byteStatusWord		: BYTE;
	strHexStatusWord	: STRING;
	iStatusWordHexa		: INT;

	xCmdFwd		: BOOL;	//Sinal digital para ligar o motor avanço
	xCmdRwd		: BOOL;	//Sinal digital para ligar o motor reverso
	iVelocidade	: INT;	//Entrada da referência de Velocidade

	iTempoIni	: INT;
	iAjuda		: INT;

	(*HearthBeat*)
	FB_HearthBeat	: FB_Ciclica;
	xHearthBeat		: BOOL;

	(*ACT00*)
	fbReadRegsETA		: FB_MBReadRegs;
	bReadRegsETA		: BOOL;
	bReadRegsBusyETA	: BOOL;
	bReadRegsErrorETA	: BOOL;
	nReadRegsErrorIdETA	: UDINT;
	nReadRegsCountETA	: UDINT;
	nQuantityETA		: WORD	:= 5;
	nMBAddrETA			: WORD	:= 3201;
	arrDataETA			: ARRAY[1..5] OF WORD;

	(*ACT01*)
	fbReadRegsVEL		: FB_MBReadRegs;
	bReadRegsVEL		: BOOL;
	bReadRegsBusyVEL	: BOOL;
	bReadRegsErrorVEL	: BOOL;
	nReadRegsErrorIdVEL	: UDINT;
	nReadRegsCountVEL	: UDINT;
	nQuantityVEL		: WORD	:= 2;
	nMBAddrVEL			: WORD	:= 8604;
	arrDataVEL			: ARRAY[1..2] OF WORD;

	(*ACT02*)
	fbWriteSingleReg	: FB_MBWriteSingleReg;
	bWriteReg			: BOOL;
	bWriteRegBusy		: BOOL;
	bWriteRegError		: BOOL;
	nWriteRegErrorId	: UDINT;
	nMBAddrWr			: WORD := 8501;
	nWrControlWord		: WORD;

	(*ACT03*)
	fbWriteSingleRegVel	: FB_MBWriteSingleReg;
	bWriteRegVel		: BOOL;
	bWriteRegBusyVel	: BOOL;
	bWriteRegErrorVel	: BOOL;
	nWriteRegErrorIdVel	: UDINT;
	nMBAddrWrVel		: WORD := 8602;
	nValueVel			: WORD;
	iVelocidadeAntiga	: INT;

	(*
(*ACT04*)
   fbReadRegsCOR     	: FB_MBReadRegs;
   bReadRegsCOR         : BOOL;
   bReadRegsBusyCOR     : BOOL;
   bReadRegsErrorCOR    : BOOL;
   nReadRegsErrorIdCOR  : UDINT;
   nReadRegsCountCOR    : UDINT;
   nQuantityCOR         : WORD:=2;
   nMBAddrCOR           : WORD:=3204;
   arrDataCOR           : ARRAY [1..2] OF WORD;
   *)
	(*ACT04*)
	fbReadRegsLastError			: FB_MBReadRegs;
	bReadRegsLastError			: BOOL;
	bReadRegsBusyLastError		: BOOL;
	bReadRegsErrorLastError		: BOOL;
	nReadRegsErrorIdLastError	: UDINT;
	nReadRegsCountLastError		: UDINT;
	nQuantityLastError			: WORD	:= 2;
	nMBAddrLastError			: WORD	:= 7121;
	arrDatanMBAddrLastError		: ARRAY[1..2] OF WORD;

	(*ACT05*)
	fbReadRegsETA_UINT			: FB_MBReadRegs;
	bReadRegsETA_UINT			: BOOL;
	bReadRegsBusyETA_UINT		: BOOL;
	bReadRegsErrorETA_UINT		: BOOL;
	nReadRegsErrorIdETA_UINT	: UDINT;
	nReadRegsCountETA_UINT		: UDINT;
	nQuantityETA_UINT			: WORD	:= 4;
	nMBAddrETA_UINT				: WORD	:= 3205;
	arrDataETA_UINT				: ARRAY[1..5] OF UINT;

	(*ACT06*)
	fbReadRegsMotorTherm		: FB_MBReadRegs;
	bReadRegsMotorTherm			: BOOL;
	bReadRegsBusyMotorTherm		: BOOL;
	bReadRegsErrorMotorTherm	: BOOL;
	nReadRegsErrorIdMotorTherm	: UDINT;
	nReadRegsCountMotorTherm	: UDINT;
	nQuantityMotorTherm			: WORD	:= 2;
	nMBAddrMotorTherm			: WORD	:= 9630;
	arrDatanMBAddrMotorTherm	: ARRAY[1..2] OF UINT;

	(*ACT07*)
	fbReadRegsMotorRunTime			: FB_MBReadRegs;
	bReadRegsMotorRunTime			: BOOL;
	bReadRegsBusyMotorRunTime		: BOOL;
	bReadRegsErrorMotorRunTime		: BOOL;
	nReadRegsErrorIdMotorRunTime	: UDINT;
	nReadRegsCountMotorRunTime		: UDINT;
	nQuantityMotorRunTime			: WORD	:= 3;
	nMBAddrMotorRunTime				: WORD	:= 3244;
	arrDatanMBAddrMotorRunTime		: ARRAY[1..3] OF UINT;

	(*ACT08*)
	fbReadRegsStoStatus			: FB_MBReadRegs;
	bReadRegsStoStatus			: BOOL;
	bReadRegsBusyStoStatus		: BOOL;
	bReadRegsErrorStoStatus		: BOOL;
	nReadRegsErrorIdStoStatus	: UDINT;
	nReadRegsCountStoStatus		: UDINT;
	nQuantityStoStatus			: WORD	:= 3;
	nMBAddrStoStatus			: WORD	:= 15322;
	arrDatanMBAddrStoStatus		: ARRAY[1..3] OF WORD;

	(*ACT09*)
	fbReadRegsAPPS			: FB_MBReadRegs;
	bReadRegsAPPS			: BOOL;
	bReadRegsBusyAPPS		: BOOL;
	bReadRegsErrorAPPS		: BOOL;
	nReadRegsErrorIdAPPS	: UDINT;
	nReadRegsCountAPPS		: UDINT;
	nQuantityAPPS			: WORD	:= 1;
	nMBAddrAPPS				: WORD	:= 15980;
	arrDatanMBAddAPPS		: ARRAY[1..2] OF WORD;

	(*Start na máquina de estados*)
	rtEnable			: R_TRIG;
	xAuxTempoContando	: BOOL;
	xAuxInversorOffline	: BOOL := FALSE;
	tonInversorOffline	: TON;
	rtReadError			: R_TRIG;
	ftReadError			: F_TRIG;
	uiStatusWord		: UINT; //Status Word que vem do inversor ATV320	

	Contador1				: CTU;
	Contador2				: CTU;
	Contador3				: CTU;
	wcont1					: WORD;
	wcont2					: WORD;
	wcont3					: WORD;
	FB_AnimaMotor			: FB_AnimaMotor;
	rtFalhanaPartida		: R_TRIG;
	rtSucessonaPartida		: R_TRIG;
	rtDisjuntorDesarmado	: R_TRIG;

	rtTrocouManAuto	: R_TRIG;
	ftTrocouManAuto	: F_TRIG;

	rtNotOnline			: R_TRIG;
	tonOnline			: TON;
	xAuxNotOnline		: BOOL;
	ftInversorOnline	: F_TRIG;

END_VAR

IF xEnable THEN

	rtEnable.CLK	:= xEnable;
	xEnabled		:= TRUE;
	xResetInversor	:= xResetDrive;
	ACT_HearthBeat();
	ACT_00_LeituraETA_CIA402();
	ACT_01_LeituraVelocidadeAtual();
	ACT_02_EscritaControlWord();
	ACT_03_EscritaVelocidade();
	ACT_04_Leitura_Last_error();
	ACT_05_LeituraETA_UINT();
	ACT_06_Leitura_Motor_Therm();
	ACT_07_Leitura_Motor_run_time();
	ACT_08_Leitura_Sto_Status();
	ACT_09_Leitura_APPS();

	uiStatusWord := WORD_TO_UINT(arrDataETA[1]);

	uiFBState				:= 1;
	bReadRegsETA			:= xHearthBeat;
	bReadRegsVEL			:= xHearthBeat;
	bWriteRegVel			:= xHearthBeat;
	bReadRegsLastError		:= xHearthBeat;
	bReadRegsETA_UINT		:= xHearthBeat;
	bReadRegsMotorTherm		:= xHearthBeat;
	bReadRegsMotorRunTime	:= xHearthBeat;
	bReadRegsStoStatus		:= xHearthBeat;
	bReadRegsAPPS			:= xHearthBeat;

	(*Se o Nó estiver ativo, e sem falhas, energiza a potência do Drive*)
	IF rtEnable.Q THEN
		iMachineState := 0;
	END_IF

	(*Converte valor da Status Word para Hexa*)
	byteStatusWord		:= UINT_TO_BYTE(uiStatusWord);
	strHexStatusWord	:= BYTE_TO_HEXSTR(in := byteStatusWord, iPrecision := 2, bLoCase := FALSE);
	iStatusWordHexa		:= STRING_TO_INT(strHexStatusWord);
	iStsWordHexa		:= iStatusWordHexa;
	(*---FIM---*)

	IF iStatusWordHexa = 17 AND NOT iMachineState = 4 THEN //535
		uiControlWord	:= 0;
		bWriteReg		:= TRUE;

		IF iStatusWordHexa = 50 THEN
			bWriteReg := FALSE;
		END_IF
	END_IF

	// INICIO CONTROLE AUTOMATICO MANUAL

	rtTrocouManAuto(CLK := xAutomaticoManual, Q =>);
	ftTrocouManAuto(CLK := xAutomaticoManual, Q =>);

	IF rtTrocouManAuto.Q OR ftTrocouManAuto.Q THEN
		xCmdFWD	:= FALSE;
		xCmdRwd	:= FALSE;
	END_IF

	IF xEmergencia THEN
		IF xLiberadoOperar THEN
			IF ((xContatoInversor OR xBypassContatoInversor) AND (xDisjuntorMOTOR OR xBypassDisjuntorMOTOR)) THEN
				IF xAutomaticoManual THEN
					IF xLigaAuto THEN
						IF xSentidoReverso THEN
							xCmdRwd := TRUE;
						ELSE
							xCmdFWD := TRUE;
						END_IF
					END_IF

					IF xDesligaAuto THEN
						xCmdFWD	:= FALSE;
						xCmdRwd	:= FALSE;
					END_IF

					iVelocidade := iSetPoinAuto;
				ELSE // manual
					IF xLigaManu THEN
						IF xSentidoReverso THEN
							xCmdRwd := TRUE;
						ELSE
							xCmdFWD := TRUE;
						END_IF
					END_IF

					IF xDesligaManu THEN
						xCmdFWD	:= FALSE;
						xCmdRwd	:= FALSE;
					END_IF

					iVelocidade := iSetPoinManu;
				END_IF
			ELSE
				xCmdFWD	:= FALSE;
				xCmdRwd	:= FALSE;
			END_IF
		ELSE
			xCmdFWD	:= FALSE;
			xCmdRwd	:= FALSE;
		END_IF
	ELSE
		xCmdFWD	:= FALSE;
		xCmdRwd	:= FALSE;
	END_IF

	// FINAL  CONTROLE AUTOMATICO MANUAL

	iTargetVelocity		:= iVelocidade;
	iVelocidadeAtual	:= WORD_TO_INT(arrDataVEL[1]);
	rCorrenteAtual		:= (WORD_TO_REAL(arrDataETA[4])) / 10;

	rVelocidadeAtualHZ := (WORD_TO_REAL(arrDataETA[2])) / 10;

	iMotorTorqueAtual := WORD_TO_INT(arrDataETA[5]);

	iMotorVoltagemAtual := UINT_TO_INT(arrDataETA_UINT[4]);

	rVoltagemEntrada := UINT_TO_REAL(arrDataETA_UINT[3]) / 10;

	rTemperaturaInversor := UINT_TO_REAL(arrDataETA_UINT[5]);

	iLastError := WORD_TO_INT(arrDatanMBAddrLastError[1]);

	iTemperaturaMotorAtual := UINT_TO_INT(arrDatanMBAddrMotorTherm[1]);

	iTempoMotorLigadoSempre := arrDatanMBAddrMotorRunTime[2];

	xStatusEmergencia := WORD_TO_BOOL(arrDatanMBAddrStoStatus[1]);

	CASE WORD_TO_INT(arrDatanMBAddAPPS[1]) OF

		0:
			sStatusInversor := 'Running';

		1:
			sStatusInversor := 'Stop';

		2:
			sStatusInversor := 'Oper. Local';

		3:
			sStatusInversor := 'Oper. Ethernet';

		4:
			sStatusInversor := 'Manual Mode Active';

		5:
			sStatusInversor := 'PID Active';

		6:
			sStatusInversor := 'Anti-Jam In progress';

		7:
			sStatusInversor := 'Flow limit In progress';

		8:
			sStatusInversor := 'PipeFill In progress';

		9:
			sStatusInversor := 'Jockey Pump Active';

		10:
			sStatusInversor := 'Boost In progress';

		11:
			sStatusInversor := 'Sleep Active';

		12:
			sStatusInversor := 'Priming Pump Active';

		13:
			sStatusInversor := 'InletPres Comp In progress';

	END_CASE

	IF NOT xInversorOnline THEN
		sStatusInversor := 'Offline';
	END_IF

	IF ((iMotorVoltagemAtual > 0.1) AND NOT xAuxTempoContando) THEN

		iTempoIni			:= UINT_TO_INT(iTempoMotorLigadoSempre);
		xAuxTempoContando	:= TRUE;

	END_IF

	IF (iMotorVoltagemAtual < 0.1 AND xAuxTempoContando) THEN

		tTempoLigadoAgora	:= T#0S;
		xAuxTempoContando	:= FALSE;

	END_IF

	//tTempoLigadoAgora := SECOND_TO_TIME((UINT_TO_INT( iTempoMotorLigadoSempre) - iTempoIni));

	nValueVel := INT_TO_WORD(iTargetVelocity);

	CASE iMachineState OF

		0:															//NST
			IF iStatusWordHexa = 50 OR iStatusWordHexa = 40 THEN	//592
				uiControlWord	:= 6;								//Com o inversor em NST, joga o inversor para 'RDY'
				bWriteReg		:= TRUE;
			END_IF

			IF iStatusWordHexa = 31 OR iStatusWordHexa = 21 THEN //561
				bWriteReg		:= FALSE;
				iMachineState	:= 1; //com o inveror em RDY joga para o passo de ativação do comando
			END_IF

			IF iStatusWordHexa = 33 THEN //563 ou 591
				bWriteReg		:= FALSE;
				iMachineState	:= 2; //com o inveror em RDY e ativado joga para o passo de comando
			END_IF

		1:							//RDY
			uiControlWord	:= 7;	//Com o inversor em RDY, Ativa o Comando
			bWriteReg		:= TRUE;

			IF iStatusWordHexa = 33 THEN //563 ou 591
				bWriteReg		:= FALSE;
				iMachineState	:= 2; //com o inveror em RDY e ativado joga para o passo de comando
			END_IF

			IF iStatusWordHexa = 50 THEN
				iMachineState := 0;
			END_IF

		2: //

			IF iStatusWordHexa = 50 THEN
				iMachineState := 0;
			END_IF

			IF uiControlWord = 15 AND iStatusWordHexa = 33 AND NOT xCmdFwd THEN
				iMachineState := 1;
			END_IF

			IF xCmdFwd THEN
				uiControlWord	:= 15; //Comando de marcha avanço
				bWriteReg		:= TRUE;

				IF iStatusWordHexa = 37 THEN
					bWriteReg		:= FALSE;
					iMachineState	:= 3;
				END_IF
			END_IF

			IF xCmdRwd THEN
				uiControlWord	:= 2063; //Comando de marcha avanço
				bWriteReg		:= TRUE;

				IF iStatusWordHexa = 37 THEN
					bWriteReg		:= FALSE;
					iMachineState	:= 5;
				END_IF
			END_IF

		3:
			IF iStatusWordHexa = 37 THEN //1591
				IF NOT xCmdFwd THEN
					IF xTipodeParada THEN
						uiControlWord	:= 7; //Comando de parada por rampa
						bWriteReg		:= TRUE;

						IF iStatusWordHexa = 33 THEN
							bWriteReg := FALSE;
						END_IF
					ELSE
						uiControlWord	:= 6; //Comando de parada por inércia
						bWriteReg		:= TRUE;

						IF iStatusWordHexa = 31 THEN
							bWriteReg := FALSE;
						END_IF
					END_IF
				END_IF

				IF xParadaRapida THEN
					iMachineState := 4;
				END_IF
			END_IF

			IF iStatusWordHexa = 31 THEN	//561
				iMachineState := 1;			//com o inveror em RDY joga para o passo de ativação do comando
			END_IF

			IF iStatusWordHexa = 33 THEN	//563
				iMachineState := 2;			//com o inveror em RDY joga para o passo de ativação do comando
			END_IF

			IF iStatusWordHexa = 50 THEN //592
				iMachineState := 6;
			END_IF

		4:
			uiControlWord	:= 2; //Comando de parada rápida		
			bWriteReg		:= TRUE;

			IF iStatusWordHexa = 17 THEN //535
				bWriteReg		:= FALSE;
				iMachineState	:= 0;
			END_IF

		5:
			IF iStatusWordHexa = 37 THEN //34359
				IF NOT xCmdRwd THEN
					IF xTipodeParada THEN
						uiControlWord	:= 7; //Comando de parada por rampa
						bWriteReg		:= TRUE;

						IF iStatusWordHexa = 33 THEN
							bWriteReg := FALSE;
						END_IF
					ELSE
						uiControlWord	:= 6; //Comando de parada por inércia
						bWriteReg		:= TRUE;

						IF iStatusWordHexa = 31 THEN
							bWriteReg := FALSE;
						END_IF

					END_IF
				END_IF

				IF xParadaRapida THEN
					iMachineState := 4;
				END_IF
			END_IF

			IF iStatusWordHexa = 31 THEN	//561
				iMachineState := 1;			//com o inveror em RDY joga para o passo de ativação do comando
			END_IF

			IF iStatusWordHexa = 33 THEN	//563
				iMachineState := 2;			//com o inveror em RDY joga para o passo de ativação do comando
			END_IF

			IF iStatusWordHexa = 50 THEN //592
				iMachineState := 6;
			END_IF

		6:
			uiControlWord	:= 0;
			bWriteReg		:= TRUE;

			IF iStatusWordHexa = 50 THEN
				bWriteReg		:= FALSE;
				iMachineState	:= 0;
			END_IF

		ELSE
			uiControlWord	:= 0; //Comando de parada rápida	
			bWriteReg		:= TRUE;

			IF iStatusWordHexa = 50 THEN
				bWriteReg := FALSE;
			END_IF

	END_CASE

	IF xResetDrive THEN
		uiControlWord	:= 128; //Comando de reset via rede	
		bWriteReg		:= TRUE;

		IF iStatusWordHexa = 50 THEN
			bWriteReg := FALSE;
		END_IF

	END_IF

	//manda um sinal de motor rodando via rede
	IF iStatusWordHexa = 37 THEN //1591
		xMotorRUN := TRUE;
	ELSE
		xMotorRUN := FALSE;
	END_IF

	(*Alterei aqui em 22/01*)
	IF iStatusWordHexa = 50 THEN
		xMotorRUN := FALSE;

		IF xResetDrive THEN
			uiControlWord	:= 128; //Comando de reset via rede	
			bWriteReg		:= TRUE;

			IF iStatusWordHexa = 31 THEN
				bWriteReg := FALSE;
			END_IF
			(*FIM*)
		END_IF
	END_IF

	nWrControlWord := UINT_TO_WORD(uiControlWord);

ELSE
	uiControlWord	:= 0;
	bWriteReg		:= TRUE;

	IF iStatusWordHexa = 50 THEN
		bWriteReg := FALSE;
	END_IF

	xEnabled		:= FALSE;
	uiFBState		:= 999;
	iMachineState	:= 0;
END_IF

//Copia sinal de liga para a saída do bloco
xCMDFwds := xCmdFWD;

//Monitora se o inversor está online

IF NOT bReadRegsErrorETA
		OR NOT bReadRegsErrorVEL
		OR NOT bReadRegsErrorLastError
		OR NOT bReadRegsErrorETA_UINT
		OR NOT bReadRegsErrorMotorTherm
		OR NOT bReadRegsErrorMotorRunTime
		OR NOT bReadRegsErrorStoStatus
		OR NOT bReadRegsErrorAPPS THEN
	xAuxNotOnline := FALSE;
ELSE
	xAuxNotOnline := TRUE;
END_IF

rtNotOnline(CLK := xAuxNotOnline, Q =>);
tonOnline(IN := NOT xAuxNotOnline, PT := T#3S, Q =>, ET =>);

IF rtNotOnline.Q THEN
	xInversorOnline := FALSE;
ELSIF tonOnline.Q THEN
	xInversorOnline := TRUE;
END_IF

ftInversorOnline(CLK := xInversorOnline, Q =>);

IF ftInversorOnline.Q THEN
	xCmdFwd	:= FALSE;
	xCmdrwd	:= FALSE;
END_IF

//Traduz a word para apresentação mais facil

CASE iStsWordHexa OF
	31:
		sWordTraduzida		:= 'NST';
		xInversoremFalha	:= TRUE;

	33:
		sWordTraduzida		:= 'RDY';
		xInversoremFalha	:= FALSE;

	37:
		sWordTraduzida		:= 'RUN';
		xInversoremFalha	:= FALSE;

	38:
		sWordTraduzida		:= 'Falha';
		xInversoremFalha	:= TRUE;

	50:
		sWordTraduzida		:= 'STO / Emergencia';
		xInversoremFalha	:= TRUE;
END_CASE

IF (NOT xCmdFwd) AND xEmergencia THEN
	iStsMotor := 1;
END_IF

IF (xCmdFwd) AND xEmergencia THEN
	iStsMotor := 2;
END_IF

rtSucessonaPartida(CLK := (iStsMotor = 2), Q =>);

Contador2
	(
		CU := rtSucessonaPartida.Q,
			RESET := xResetRegistros,
			PV :=,
			Q =>,
			CV => wcont2);

IF (NOT xDisjuntorMOTOR) AND (NOT xBypassDisjuntorMOTOR) THEN
	iStsMotor := 3;
END_IF

rtDisjuntorDesarmado(CLK := iStsMotor = 3, Q =>);

Contador1
	(
		CU := rtDisjuntorDesarmado.Q,
			RESET := xResetRegistros,
			PV :=,
			Q =>,
			CV => wcont1);

IF iStsWordHexa = 38 OR NOT xInversorOnline THEN
	iStsMotor := 5;
END_IF

rtFalhanaPartida(CLK := iStsMotor = 5, Q =>);

Contador3
	(
		CU := rtFalhanaPartida.Q,
			RESET := xResetRegistros,
			PV :=,
			Q =>,
			CV => wcont3);

IF NOT xLiberadoOperar THEN
	iStsMotor := 6;
END_IF

IF NOT xEmergencia THEN
	iStsMotor := 4;
END_IF

iDisjDesarm			:= WORD_TO_INT(wcont1);
iPartidas			:= WORD_TO_INT(wcont2);
iInversoremFalha	:= WORD_TO_INT(wcont3);

//FB_AnimaMotor(iStsMotor:= iStsMotor, dwStateColor=> dwStateColor);

ACTION ACT_00_LeituraETA_CIA402:
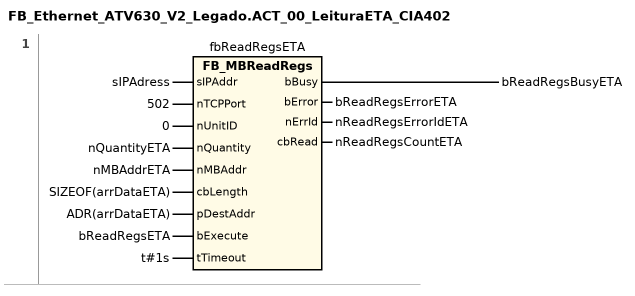
// NETWORK 1
fbReadRegsETA(
    sIPAddr := sIPAdress,
    nTCPPort := 502,
    nUnitID := 0,
    nQuantity := nQuantityETA,
    nMBAddr := nMBAddrETA,
    cbLength := SIZEOF(arrDataETA),
    pDestAddr := ADR(arrDataETA),
    bExecute := bReadRegsETA,
    tTimeout := t#1s,
    bError => bReadRegsErrorETA,
    nErrId => nReadRegsErrorIdETA,
    cbRead => nReadRegsCountETA); // FB_MBReadRegs
bReadRegsBusyETA := fbReadRegsETA.bBusy;
END_ACTION

ACTION ACT_01_LeituraVelocidadeAtual:
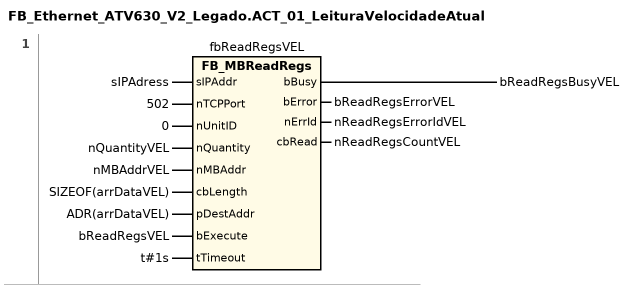
// NETWORK 1
fbReadRegsVEL(
    sIPAddr := sIPAdress,
    nTCPPort := 502,
    nUnitID := 0,
    nQuantity := nQuantityVEL,
    nMBAddr := nMBAddrVEL,
    cbLength := SIZEOF(arrDataVEL),
    pDestAddr := ADR(arrDataVEL),
    bExecute := bReadRegsVEL,
    tTimeout := t#1s,
    bError => bReadRegsErrorVEL,
    nErrId => nReadRegsErrorIdVEL,
    cbRead => nReadRegsCountVEL); // FB_MBReadRegs
bReadRegsBusyVEL := fbReadRegsVEL.bBusy;
END_ACTION

ACTION ACT_03_EscritaVelocidade:
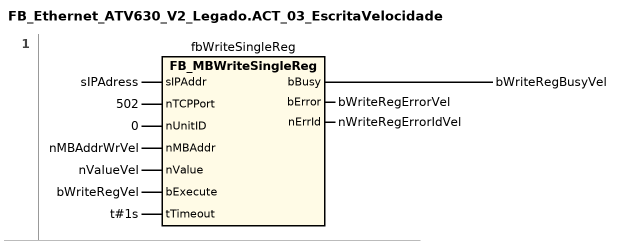
// NETWORK 1
fbWriteSingleReg(
    sIPAddr := sIPAdress,
    nTCPPort := 502,
    nUnitID := 0,
    nMBAddr := nMBAddrWrVel,
    nValue := nValueVel,
    bExecute := bWriteRegVel,
    tTimeout := t#1s,
    bError => bWriteRegErrorVel,
    nErrId => nWriteRegErrorIdVel); // FB_MBWriteSingleReg
bWriteRegBusyVel := fbWriteSingleReg.bBusy;
END_ACTION

ACTION ACT_04_Leitura_Last_error:
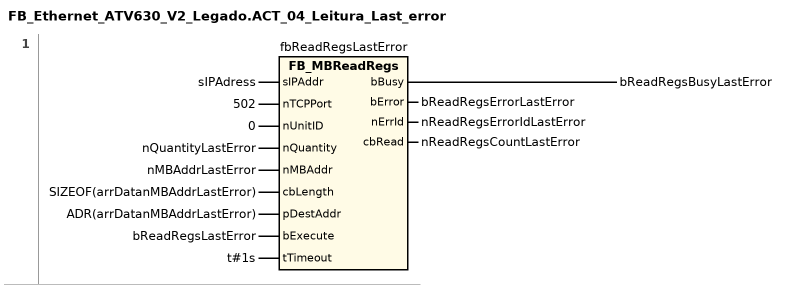
// NETWORK 1
fbReadRegsLastError(
    sIPAddr := sIPAdress,
    nTCPPort := 502,
    nUnitID := 0,
    nQuantity := nQuantityLastError,
    nMBAddr := nMBAddrLastError,
    cbLength := SIZEOF(arrDatanMBAddrLastError),
    pDestAddr := ADR(arrDatanMBAddrLastError),
    bExecute := bReadRegsLastError,
    tTimeout := t#1s,
    bError => bReadRegsErrorLastError,
    nErrId => nReadRegsErrorIdLastError,
    cbRead => nReadRegsCountLastError); // FB_MBReadRegs
bReadRegsBusyLastError := fbReadRegsLastError.bBusy;
END_ACTION

ACTION ACT_05_LeituraETA_UINT:
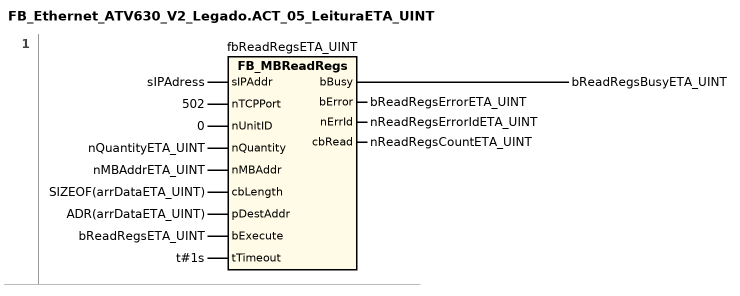
// NETWORK 1
fbReadRegsETA_UINT(
    sIPAddr := sIPAdress,
    nTCPPort := 502,
    nUnitID := 0,
    nQuantity := nQuantityETA_UINT,
    nMBAddr := nMBAddrETA_UINT,
    cbLength := SIZEOF(arrDataETA_UINT),
    pDestAddr := ADR(arrDataETA_UINT),
    bExecute := bReadRegsETA_UINT,
    tTimeout := t#1s,
    bError => bReadRegsErrorETA_UINT,
    nErrId => nReadRegsErrorIdETA_UINT,
    cbRead => nReadRegsCountETA_UINT); // FB_MBReadRegs
bReadRegsBusyETA_UINT := fbReadRegsETA_UINT.bBusy;
END_ACTION

ACTION ACT_06_Leitura_Motor_Therm:
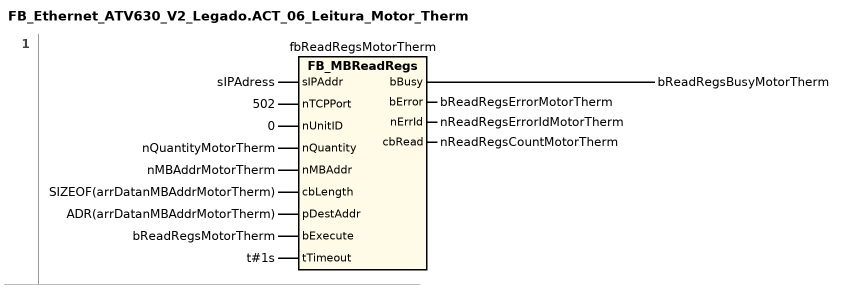
// NETWORK 1
fbReadRegsMotorTherm(
    sIPAddr := sIPAdress,
    nTCPPort := 502,
    nUnitID := 0,
    nQuantity := nQuantityMotorTherm,
    nMBAddr := nMBAddrMotorTherm,
    cbLength := SIZEOF(arrDatanMBAddrMotorTherm),
    pDestAddr := ADR(arrDatanMBAddrMotorTherm),
    bExecute := bReadRegsMotorTherm,
    tTimeout := t#1s,
    bError => bReadRegsErrorMotorTherm,
    nErrId => nReadRegsErrorIdMotorTherm,
    cbRead => nReadRegsCountMotorTherm); // FB_MBReadRegs
bReadRegsBusyMotorTherm := fbReadRegsMotorTherm.bBusy;
END_ACTION

ACTION ACT_07_Leitura_Motor_run_time:
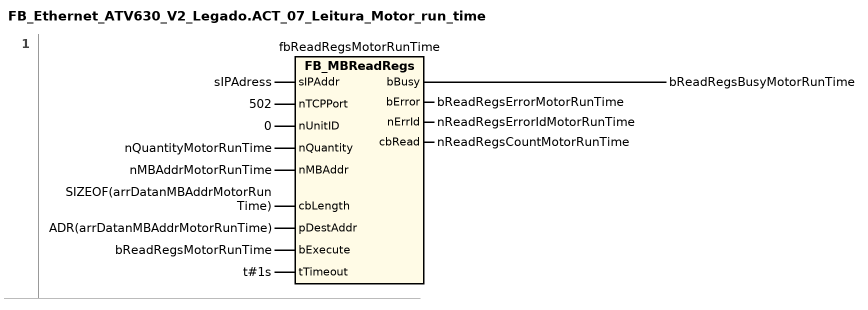
// NETWORK 1
fbReadRegsMotorRunTime(
    sIPAddr := sIPAdress,
    nTCPPort := 502,
    nUnitID := 0,
    nQuantity := nQuantityMotorRunTime,
    nMBAddr := nMBAddrMotorRunTime,
    cbLength := SIZEOF(arrDatanMBAddrMotorRunTime),
    pDestAddr := ADR(arrDatanMBAddrMotorRunTime),
    bExecute := bReadRegsMotorRunTime,
    tTimeout := t#1s,
    bError => bReadRegsErrorMotorRunTime,
    nErrId => nReadRegsErrorIdMotorRunTime,
    cbRead => nReadRegsCountMotorRunTime); // FB_MBReadRegs
bReadRegsBusyMotorRunTime := fbReadRegsMotorRunTime.bBusy;
END_ACTION

ACTION ACT_08_Leitura_Sto_Status:
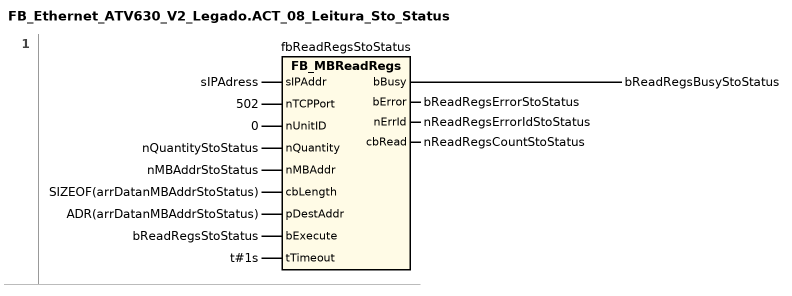
// NETWORK 1
fbReadRegsStoStatus(
    sIPAddr := sIPAdress,
    nTCPPort := 502,
    nUnitID := 0,
    nQuantity := nQuantityStoStatus,
    nMBAddr := nMBAddrStoStatus,
    cbLength := SIZEOF(arrDatanMBAddrStoStatus),
    pDestAddr := ADR(arrDatanMBAddrStoStatus),
    bExecute := bReadRegsStoStatus,
    tTimeout := t#1s,
    bError => bReadRegsErrorStoStatus,
    nErrId => nReadRegsErrorIdStoStatus,
    cbRead => nReadRegsCountStoStatus); // FB_MBReadRegs
bReadRegsBusyStoStatus := fbReadRegsStoStatus.bBusy;
END_ACTION

ACTION ACT_09_Leitura_APPS:
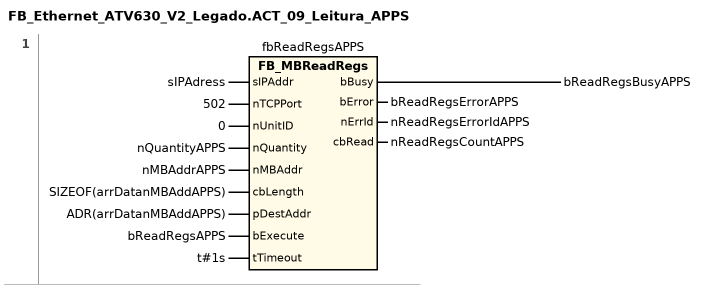
// NETWORK 1
fbReadRegsAPPS(
    sIPAddr := sIPAdress,
    nTCPPort := 502,
    nUnitID := 0,
    nQuantity := nQuantityAPPS,
    nMBAddr := nMBAddrAPPS,
    cbLength := SIZEOF(arrDatanMBAddAPPS),
    pDestAddr := ADR(arrDatanMBAddAPPS),
    bExecute := bReadRegsAPPS,
    tTimeout := t#1s,
    bError => bReadRegsErrorAPPS,
    nErrId => nReadRegsErrorIdAPPS,
    cbRead => nReadRegsCountAPPS); // FB_MBReadRegs
bReadRegsBusyAPPS := fbReadRegsAPPS.bBusy;
END_ACTION

ACTION ACT_HearthBeat:
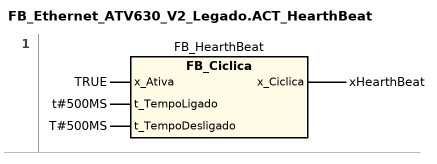
// NETWORK 1
FB_HearthBeat(x_Ativa := TRUE, t_TempoLigado := t#500MS, t_TempoDesligado := T#500MS); // FB_Ciclica
xHearthBeat := FB_HearthBeat.x_Ciclica;
END_ACTION

END_FUNCTION_BLOCK

// Legado/FB_PartidaDireta_V2_Legado
FUNCTION_BLOCK FB_PartidaDireta_V2_Legado
VAR_INPUT
	xEnable					: BOOL;
	xContatorLigado			: BOOL;					(*Status da contatora ou do drive de que o motor partiu*)
	xByPassContator			: BOOL;					//Sinal de by pass do contato da contatora
	xDisjuntorOK			: BOOL;					(*Status do disjuntor motor*)
	xByPassDisjuntor		: BOOL;					//Sinal de by pass do contato do disjuntor
	xLiberadoOperar			: BOOL;					//Sinal de Bloqueio
	iSetPoinAuto			: INT;					// velocidadde que sera mandada para o bloco de comunicação
	iSetPoinManu			: INT;					// velocidadde que sera mandada para o bloco de comunicação
	xLigaAuto				: BOOL;					// liga inversor em automatico
	xDesligaAuto			: BOOL;					// Desliga inversor em automatico
	xLigaManu				: BOOL;					// liga inversor em manual
	xDesligaManu			: BOOL;					// Desliga inversor em manual
	xAutomaticoManual		: BOOL;					// se automatico = true se manual = false
	xReset					: BOOL;					(*Sinal para resetar as falhas*)
	xEmergenciaOK			: BOOL;					(*Sinal de Emergência*)
	xResetRegistros			: BOOL;					(*Sinal apra resetar os contadores e registradores*)
	tTempoFeedBackContator	: TIME := T#1S500MS;	(*Tempo entre acionar a Saída e receber o FeedBack da Contatora*)
END_VAR
VAR_OUTPUT
	xEnabled		: BOOL;
	xCmdFwd			: BOOL;	(*Liga Motor pra frente*)
	iVelocidade		: INT;	// velocidade para bloco de comunicação
	iStsMotor		: INT;	(*Status da Partida 1=Parado 2=Ligado 3=Disjuntor Desarmado 4=Emergência 5=Falha na Partida 6=Bloqueado 999=Bloco desabilitado*)
	xResetDrive		: BOOL;	// sinal para o drive dar reset
	xPartidaOK		: BOOL;	(*Status de partida Ligada*)
	xPartidaemFalha	: BOOL;	(*Status de partida em falha*)
	xFalhaPartida	: BOOL;	(*Se o comando de partida foi dado mas o status não chegou*)
	iDisjDesarm		: INT;	(*Contagem do numero de desarmes do disjuntor*)
	iPartidas		: INT;	(*Contagem do numero de partidas com sucesso do bloco*)
	iFalhaPartida	: INT;	(*Contagem do numero de falhas na partida do bloco*)
	dwStateColor	: DWORD;
END_VAR
VAR
	xImpedePartida			: BOOL;
	TON_Partida				: TON;
	ET_Partida				: TIME;
	Contador1				: CTU;
	Contador2				: CTU;
	Contador3				: CTU;
	wcont1					: WORD;
	wcont2					: WORD;
	wcont3					: WORD;
	rtFalhanaPartida		: R_TRIG;
	rtSucessonaPartida		: R_TRIG;
	rtDisjuntorDesarmado	: R_TRIG;
	//FB_AnimaMotor : FB_AnimaMotor;
	xDisjuntorEmFalha : BOOL;
END_VAR

// controle das entradas
IF xEnable THEN
	xEnabled := TRUE;

	// INICIO CONTROLE AUTOMATICO MANUAL
	IF xEmergenciaOK THEN
		IF xLiberadoOperar THEN
			IF ((NOT xFalhaPartida) AND (xDisjuntorOK OR xByPassDisjuntor)) THEN
				IF xAutomaticoManual THEN //Automatico
					IF xLigaAuto THEN
						xCmdFWD := TRUE;
					END_IF

					IF xDesligaAuto THEN
						xCmdFWD := FALSE;
					END_IF

					iVelocidade := iSetPoinAuto;
				ELSE // manual
					IF xLigaManu THEN
						xCmdFWD := TRUE;
					END_IF

					IF xDesligaManu THEN
						xCmdFWD := FALSE;
					END_IF

					iVelocidade := iSetPoinManu;
				END_IF
			ELSE
				xCmdFWD := FALSE;
			END_IF
		ELSE
			xCmdFWD := FALSE;
		END_IF
	ELSE
		xCmdFWD := FALSE;
	END_IF

	// FINAL  CONTROLE AUTOMATICO MANUAL

	xResetDrive := xReset;

	TON_Partida(IN := (xCmdFwd) AND NOT (xContatorLigado OR xByPassContator), PT := tTempoFeedBackContator, Q =>, ET => ET_Partida);

	IF TON_Partida.q THEN
		xFalhaPartida := TRUE;
	END_IF

	IF xReset THEN
		xFalhaPartida := FALSE;
	END_IF

	IF (NOT xCmdFwd) AND NOT xImpedePartida AND xEmergenciaOK THEN
		iStsMotor := 1;
	END_IF

	IF (xCmdFwd) AND (NOT xImpedePartida OR xEmergenciaOK) THEN
		iStsMotor := 2;
	END_IF

	rtSucessonaPartida(CLK := (iStsMotor = 2 AND (xContatorLigado OR xByPassContator)), Q =>);

	Contador2
		(
			CU := rtSucessonaPartida.Q,
				RESET := xResetRegistros,
				PV :=,
				Q =>,
				CV => wcont2);

	IF (NOT xDisjuntorOK) THEN
		iStsMotor := 3;
	END_IF

	rtDisjuntorDesarmado(CLK := iStsMotor = 3, Q =>);

	Contador1
		(
			CU := rtDisjuntorDesarmado.Q,
				RESET := xResetRegistros,
				PV :=,
				Q =>,
				CV => wcont1);

	IF xFalhaPartida THEN
		iStsMotor := 5;
	END_IF

	rtFalhanaPartida(CLK := iStsMotor = 5, Q =>);

	Contador3
		(
			CU := rtFalhanaPartida.Q,
				RESET := xResetRegistros,
				PV :=,
				Q =>,
				CV => wcont3);

	IF NOT xLiberadoOperar THEN
		iStsMotor := 6;
	END_IF

	IF NOT xEmergenciaOK THEN
		iStsMotor := 4;
	END_IF

	iDisjDesarm		:= WORD_TO_INT(wcont1);
	iPartidas		:= WORD_TO_INT(wcont2);
	iFalhaPartida	:= WORD_TO_INT(wcont3);

	xDisjuntorEmFalha := NOT xDisjuntorOK AND NOT xByPassDisjuntor;

	IF (NOT xEmergenciaOK) OR (NOT xLiberadoOperar) OR (xDisjuntorEmFalha) THEN
		xPartidaemFalha := TRUE;
	ELSE
		xPartidaemFalha := FALSE;
	END_IF

	xPartidaOK := NOT xPartidaemFalha AND xCmdFwd;

ELSE
	xEnabled	:= FALSE;
	iStsMotor	:= 999;
END_IF

//FB_AnimaMotor(iStsMotor:= iStsMotor, dwStateColor=> dwStateColor);

END_FUNCTION_BLOCK

// Legado/FB_PartidaDiretaReversao_V0_Legado
FUNCTION_BLOCK FB_PartidaDiretaReversao_V0_Legado
VAR_INPUT
	xEnable					: BOOL;
	xContatorLigado			: BOOL;					(*Status da contatora ou do drive de que o motor partiu*)
	xByPassContator			: BOOL;					//Sinal de by pass do contato da contatora
	xDisjuntorOK			: BOOL;					(*Status do disjuntor motor*)
	xByPassDisjuntor		: BOOL;					//Sinal de by pass do contato do disjuntor
	xLiberadoOperar			: BOOL;					//Sinal de Bloqueio
	xLigaAutoFwd			: BOOL;					// liga Partida em automatico FWD
	xLigaAutoRwd			: BOOL;					// liga Partida em automatico FWD	
	xDesligaAuto			: BOOL;					// Desliga inversor em automatico
	xLigaManuFWD			: BOOL;					// liga inversor em manual
	xLigaManuRWD			: BOOL;					// liga inversor em manual
	xDesligaManu			: BOOL;					// Desliga inversor em manual
	xAutomaticoManual		: BOOL;					// se automatico = true se manual = false
	xReset					: BOOL;					(*Sinal para resetar as falhas*)
	xEmergencia				: BOOL;					(*Sinal de Emergência*)
	xResetRegistros			: BOOL;					(*Sinal apra resetar os contadores e registradores*)
	tTempoFeedBackContator	: TIME := T#1S500MS;	(*Tempo entre acionar a Saída e receber o FeedBack da Contatora*)
END_VAR

VAR_OUTPUT
	xEnabled		: BOOL;
	xCmdFwd			: BOOL;	(*Liga Motor pra frente*)
	xCmdRWD			: BOOL;	(*Liga Motor Reverso*)
	iStsMotor		: INT;	(*Status da Partida 1=Parado 2=Ligado 3=Disjuntor Desarmado 4=Emergência 5=Falha na Partida 6=Bloqueado 999=Bloco desabilitado*)
	xPartidaOK		: BOOL;	(*Status de partida Ligada*)
	xPartidaemFalha	: BOOL;	(*Status de partida em falha*)
	xFalhaPartida	: BOOL;	(*Se o comando de partida foi dado mas o status não chegou*)
	iDisjDesarm		: INT;	(*Contagem do numero de desarmes do disjuntor*)
	iPartidas		: INT;	(*Contagem do numero de partidas com sucesso do bloco*)
	iFalhaPartida	: INT;	(*Contagem do numero de falhas na partida do bloco*)
	dwStateColor	: DWORD;
END_VAR
VAR
	xImpedePartida			: BOOL;
	TON_Partida				: TON;
	ET_Partida				: TIME;
	Contador1				: CTU;
	Contador2				: CTU;
	Contador3				: CTU;
	wcont1					: WORD;
	wcont2					: WORD;
	wcont3					: WORD;
	rtFalhanaPartida		: R_TRIG;
	rtSucessonaPartida		: R_TRIG;
	rtDisjuntorDesarmado	: R_TRIG;
	FB_AnimaMotor			: FB_AnimaMotor;
	xDisjuntorEmFalha		: BOOL;
END_VAR


IF xEnable THEN
	xEnabled := TRUE;

	// INICIO CONTROLE AUTOMATICO MANUAL
	IF xEmergencia THEN
		IF xLiberadoOperar THEN
			IF ((NOT xFalhaPartida) AND (xDisjuntorOK OR xByPassDisjuntor)) THEN
				IF xAutomaticoManual THEN //Automatico
					IF xLigaAutoFwd THEN
						xCmdFWD := TRUE;
					END_IF

					IF xLigaAutoRwd THEN
						xCmdRWD := TRUE;
					END_IF

					IF xDesligaAuto THEN
						xCmdFWD	:= FALSE;
						xCmdRWD	:= FALSE;
					END_IF
				ELSE // manual
					IF xLigaManuFWD THEN
						xCmdFWD := TRUE;
					END_IF

					IF xLigaManuRWD THEN
						xCmdRWD := TRUE;
					END_IF

					IF xDesligaManu THEN
						xCmdFWD	:= FALSE;
						xCmdRWD	:= FALSE;
					END_IF
				END_IF
			ELSE
				xCmdFWD	:= FALSE;
				xCmdRWD	:= FALSE;
			END_IF
		ELSE
			xCmdFWD	:= FALSE;
			xCmdRWD	:= FALSE;
		END_IF
	ELSE
		xCmdFWD	:= FALSE;
		xCmdRWD	:= FALSE;
	END_IF

	// FINAL  CONTROLE AUTOMATICO MANUAL

	TON_Partida(IN := (xCmdFwd) AND NOT (xContatorLigado OR xByPassContator), PT := tTempoFeedBackContator, Q =>, ET => ET_Partida);

	IF TON_Partida.q THEN
		xFalhaPartida := TRUE;
	END_IF

	IF xReset THEN
		xFalhaPartida := FALSE;
	END_IF

	IF (NOT xCmdFwd OR NOT xCmdRWD) AND NOT xImpedePartida AND xEmergencia THEN
		iStsMotor := 1;
	END_IF

	IF (xCmdFwd OR xCmdRWD) AND (NOT xImpedePartida OR xEmergencia) THEN
		iStsMotor := 2;
	END_IF

	rtSucessonaPartida(CLK := (iStsMotor = 2 AND (xContatorLigado OR xByPassContator)), Q =>);

	Contador2
		(
			CU := rtSucessonaPartida.Q,
				RESET := xResetRegistros,
				PV :=,
				Q =>,
				CV => wcont2);

	IF (NOT xDisjuntorOK) THEN
		iStsMotor := 3;
	END_IF

	rtDisjuntorDesarmado(CLK := iStsMotor = 3, Q =>);

	Contador1
		(
			CU := rtDisjuntorDesarmado.Q,
				RESET := xResetRegistros,
				PV :=,
				Q =>,
				CV => wcont1);

	IF xFalhaPartida THEN
		iStsMotor := 5;
	END_IF

	rtFalhanaPartida(CLK := iStsMotor = 5, Q =>);

	Contador3
		(
			CU := rtFalhanaPartida.Q,
				RESET := xResetRegistros,
				PV :=,
				Q =>,
				CV => wcont3);

	IF NOT xLiberadoOperar THEN
		iStsMotor := 6;
	END_IF

	IF NOT xEmergencia THEN
		iStsMotor := 4;
	END_IF

	iDisjDesarm		:= WORD_TO_INT(wcont1);
	iPartidas		:= WORD_TO_INT(wcont2);
	iFalhaPartida	:= WORD_TO_INT(wcont3);

	xDisjuntorEmFalha := NOT xDisjuntorOK AND NOT xByPassDisjuntor;

	IF (NOT xEmergencia) OR (NOT xLiberadoOperar) OR (xDisjuntorEmFalha) THEN
		xPartidaemFalha := TRUE;
	ELSE
		xPartidaemFalha := FALSE;
	END_IF

ELSE
	xEnabled	:= FALSE;
	iStsMotor	:= 999;
END_IF

FB_AnimaMotor(iStsMotor := iStsMotor, dwStateColor => dwStateColor);

END_FUNCTION_BLOCK

// POUs/Beckhoff/AX5000/FB_Comunicacao_AX5000
FUNCTION_BLOCK FB_Comunicacao_AX5000
VAR_INPUT
	rAceleracao : REAL;
	rDesceleracao : REAL;
	rJerk : LREAL := 10000;
	stHoraAgora : TIMESTRUCT;
END_VAR
VAR_IN_OUT
	stMotor : st_Partida;
END_VAR
VAR_OUTPUT
	State			: INT :=0;
END_VAR
VAR	
	AxisREF : AXIS_REF;
	iTemperaturaInversor AT %I* : UINT;
	iTemperaturaMotor AT %I* : UINT; 
	iCorrente AT %I* : INT; 
	

	ExAxPower 		: MC_Power;
	ExAxStop 		: MC_Stop;
	ExAxReset 		: MC_Reset;
	fbSoEReset		: FB_SoEReset;
	fbMC_Halt		: MC_Halt;
	ExAxMvVelo 		: MC_MoveVelocity;
	fbMCReadStatus	: MC_ReadStatus;
	
	
	ExAxVeloReal	: MC_ReadActualVelocity;
	ExAxLeErro		: MC_ReadAxisError;
	ExAxLeTempMotor	: FB_SoEReadMotorTemperature;
	
	fbSoEReadDiagNumber:FB_SoEReadDiagNumber;
	fbSoEReadDiagMsg: 	FB_SoEReadDiagMessage;
	
	
	xResetInterno : BOOL;
	
	rtMudouVelo : R_TRIG;
	iVeloAnterior : INT;
	
	tonOnline : TON;
	
	raux : REAL;
	iAux : INT := 500;
	
	Enable_Positive : BOOL := TRUE;
	Enable_Negative : BOOL := TRUE;
	
	iBufferAbsoluteCurrent : ARRAY[0..9] OF INT;
	iCurrentIndex:			INT;
	
	xFirstScan : BOOL := TRUE;
	
	
	iEstadoLeCorrente 	: INT;
	rPCorrenteDePico 	: REAL;
	iAuxCorrenteDePico	: INT;
	fbReadCorrenteDePico: FB_SoERead;
	tonEsperaInicio		: TON;
	filtroCorrente		: FT_PT1 (*Filter_PT1*) ;	
	
	
	rtLigou : R_TRIG;
	
	
	iAceleracaoCalculada : udINT;
	iDesaceleracaoCalculada : UDINT;
	iJerkCalculado : UDINT;
	xCalcula : BOOL := TRUE;
	sAux : STRING;
	
END_VAR



stMotor.En.xTemInversor := AxisREF.NcToPlc.DcTimeStamp <> 0;


IF stMotor.En.xTemInversor THEN
	
	//update local variables from hardware
	AxisREF.ReadStatus();
	
	AxisREF.Status.ErrorID;
	
	
	rtMudouVelo(CLK:= iVeloAnterior <> stMotor.Sa.iVelocidade, Q=> );
	rtLigou(CLK:= stMotor.Sa.xCmdFwd OR stMotor.Sa.xCmdRev, Q=> );
	IF rtMudouVelo.q OR rtLigou.q THEN	
		iVeloAnterior := stMotor.Sa.iVelocidade;
		
		ExAxMvVelo.Direction := MC_Direction.MC_Positive_Direction;
		
		//Se for pro outro lado ele inverte o sentido
		IF stMotor.Sa.xCmdRev THEN
			ExAxMvVelo.Direction := MC_Direction.MC_Negative_Direction;
		END_IF
		//se tiver negativo ele deixa positivo pra nao cagar o role
		IF stMotor.Sa.iVelocidade < 0 THEN
			stMotor.Sa.iVelocidade := stMotor.Sa.iVelocidade *-1;
		END_IF
		ExAxMvVelo.Velocity := stMotor.Sa.iVelocidade * 6;
		
		
		ExAxMvVelo.Execute := FALSE;
		ExAxMvVelo(Axis := AxisREF);
	END_IF 
	
	ControlaACCDEC();
	
	
	CASE State OF
		0:	//Ativa o driver
			ExAxPower.Enable := TRUE; 
			ExAxPower.Enable_Positive := Enable_Positive;
			ExAxPower.Enable_Negative := Enable_Negative;
			State := 1;
			
